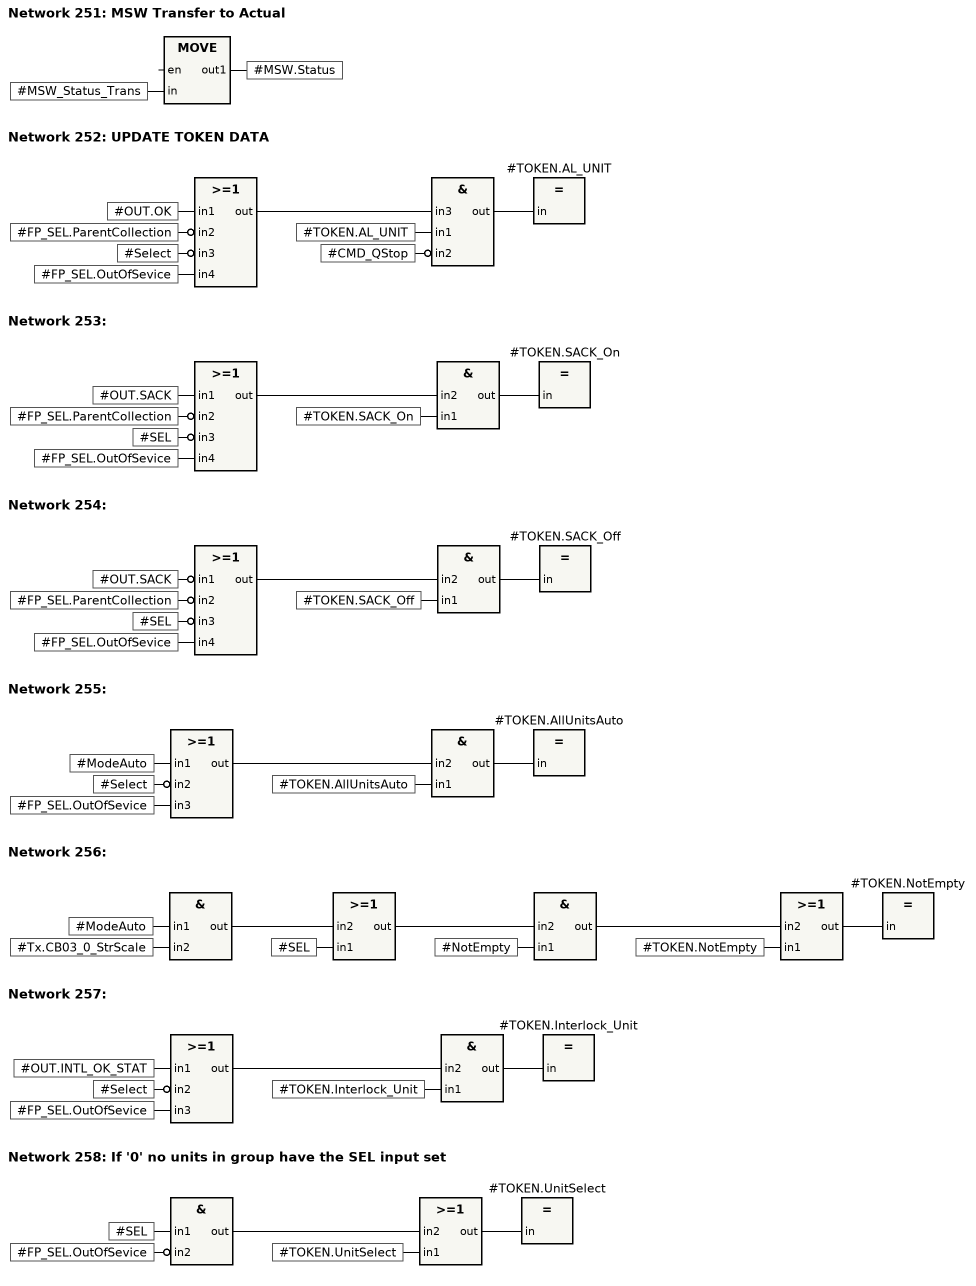
   #MSW.Status := #MSW_Status_Trans;
END_REGION

REGION Network 252: UPDATE TOKEN DATA
   #TOKEN.AL_UNIT := (#OUT.OK OR NOT #FP_SEL.ParentCollection OR NOT #Select OR #FP_SEL.OutOfSevice) AND #TOKEN.AL_UNIT AND NOT #CMD_QStop;
END_REGION

REGION Network 253
   // Build 005 - 24.Jun.2020 (MIA-US): Replace "Select" with "SEL"
   #TOKEN.SACK_On := (#OUT.SACK OR NOT #FP_SEL.ParentCollection OR NOT #SEL OR #FP_SEL.OutOfSevice) AND #TOKEN.SACK_On;
END_REGION

REGION Network 254
   #TOKEN.SACK_Off := (NOT #OUT.SACK OR NOT #FP_SEL.ParentCollection OR NOT #SEL OR #FP_SEL.OutOfSevice) AND #TOKEN.SACK_Off;
END_REGION

REGION Network 255
   #TOKEN.AllUnitsAuto := (#ModeAuto OR NOT #Select OR #FP_SEL.OutOfSevice) AND #TOKEN.AllUnitsAuto;
END_REGION

REGION Network 256
   #TOKEN.NotEmpty := (((#ModeAuto AND #Tx.CB03_0_StrScale) OR #SEL) AND #NotEmpty) OR #TOKEN.NotEmpty;
END_REGION

REGION Network 257
   #TOKEN.Interlock_Unit := (#OUT.INTL_OK_STAT OR NOT #Select OR #FP_SEL.OutOfSevice) AND #TOKEN.Interlock_Unit;
END_REGION

REGION Network 258: If '0' no units in group have the SEL input set
   #TOKEN.UnitSelect := (#SEL AND NOT #FP_SEL.OutOfSevice) OR #TOKEN.UnitSelect;
END_REGION

REGION Network 259: Start Warning
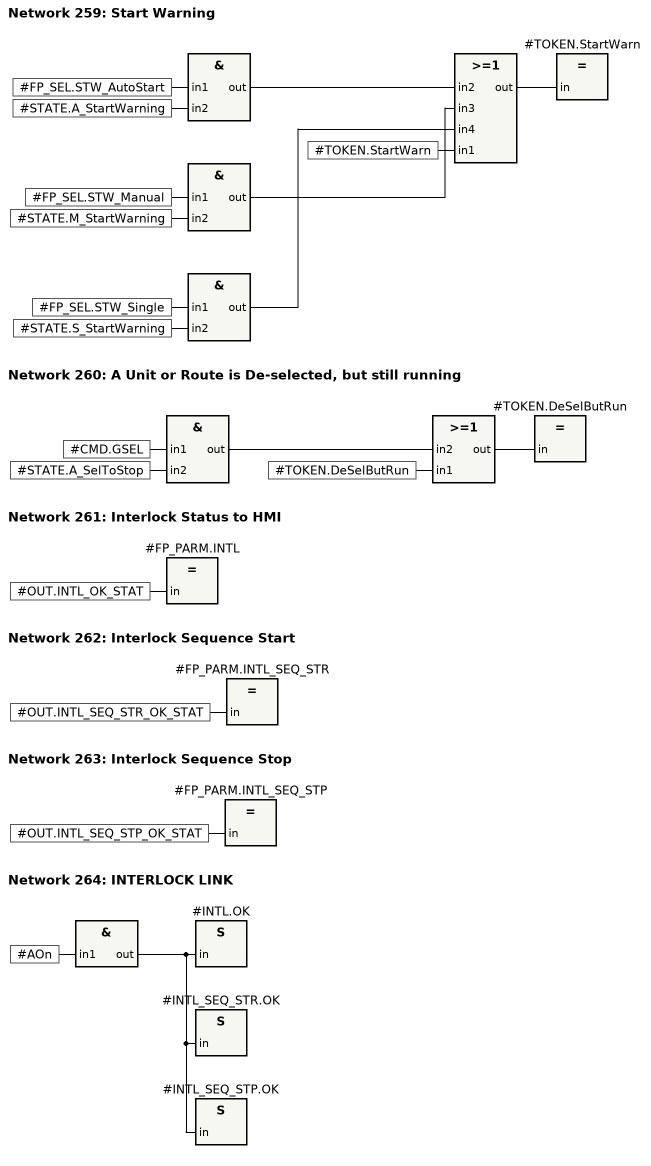
   #TOKEN.StartWarn := (#FP_SEL.STW_AutoStart AND #STATE.A_StartWarning) OR (#FP_SEL.STW_Manual AND #STATE.M_StartWarning) OR (#FP_SEL.STW_Single AND #STATE.S_StartWarning) OR #TOKEN.StartWarn;
END_REGION

REGION Network 260: A Unit or Route is De-selected, but still running
   #TOKEN.DeSelButRun := (#CMD.GSEL AND #STATE.A_SelToStop) OR #TOKEN.DeSelButRun;
END_REGION

REGION Network 261: Interlock Status to HMI
   #FP_PARM.INTL := #OUT.INTL_OK_STAT;
END_REGION

REGION Network 262: Interlock Sequence Start
   #FP_PARM.INTL_SEQ_STR := #OUT.INTL_SEQ_STR_OK_STAT;
END_REGION

REGION Network 263: Interlock Sequence Stop
   #FP_PARM.INTL_SEQ_STP := #OUT.INTL_SEQ_STP_OK_STAT;
END_REGION

REGION Network 264: INTERLOCK LINK
   IF #AOn THEN
       #INTL.OK := TRUE;
       #INTL_SEQ_STR.OK := TRUE;
       #INTL_SEQ_STP.OK := TRUE;
   END_IF;
END_REGION

REGION Network 265: Bit 1: Detect first occuring interlock, unit running
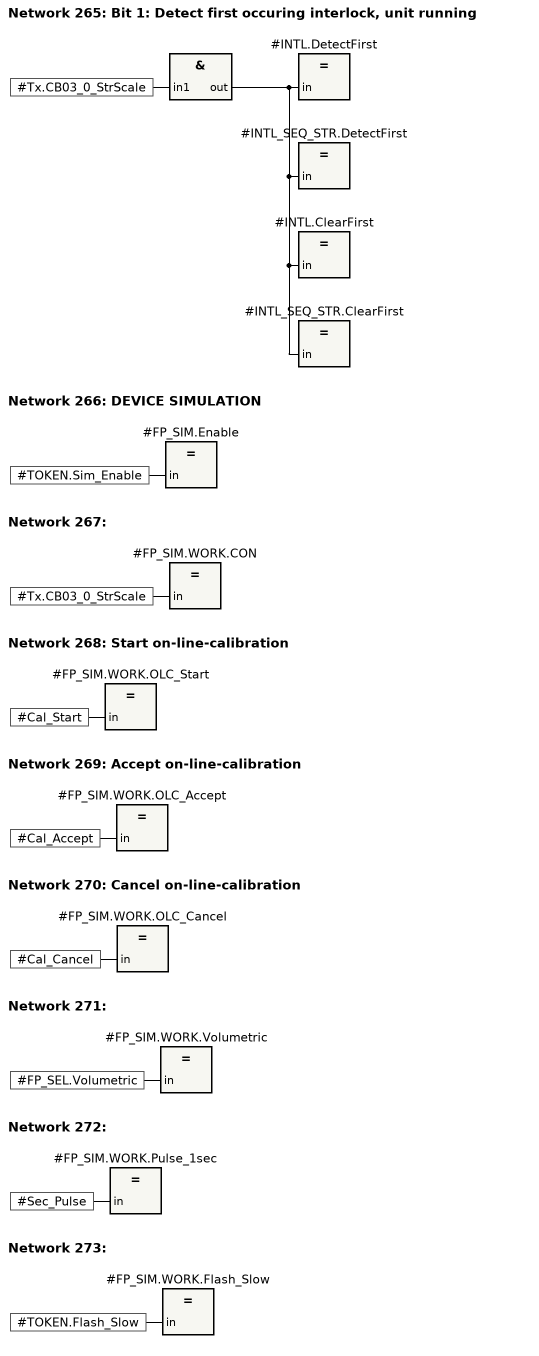
   #INTL.DetectFirst := #Tx.CB03_0_StrScale;
   #INTL_SEQ_STR.DetectFirst := #Tx.CB03_0_StrScale;
   #INTL.ClearFirst := #Tx.CB03_0_StrScale;
   #INTL_SEQ_STR.ClearFirst := #Tx.CB03_0_StrScale;
END_REGION

REGION Network 266: DEVICE SIMULATION
   #FP_SIM.Enable := #TOKEN.Sim_Enable;
END_REGION

REGION Network 267
   #FP_SIM.WORK.CON := #Tx.CB03_0_StrScale;
END_REGION

REGION Network 268: Start on-line-calibration
   #FP_SIM.WORK.OLC_Start := #Cal_Start;
END_REGION

REGION Network 269: Accept on-line-calibration
   #FP_SIM.WORK.OLC_Accept := #Cal_Accept;
END_REGION

REGION Network 270: Cancel on-line-calibration
   #FP_SIM.WORK.OLC_Cancel := #Cal_Cancel;
END_REGION

REGION Network 271
   #FP_SIM.WORK.Volumetric := #FP_SEL.Volumetric;
END_REGION

REGION Network 272
   #FP_SIM.WORK.Pulse_1sec := #Sec_Pulse;
END_REGION

REGION Network 273
   #FP_SIM.WORK.Flash_Slow := #TOKEN.Flash_Slow;
END_REGION

REGION Network 274: Write STAT to OUT
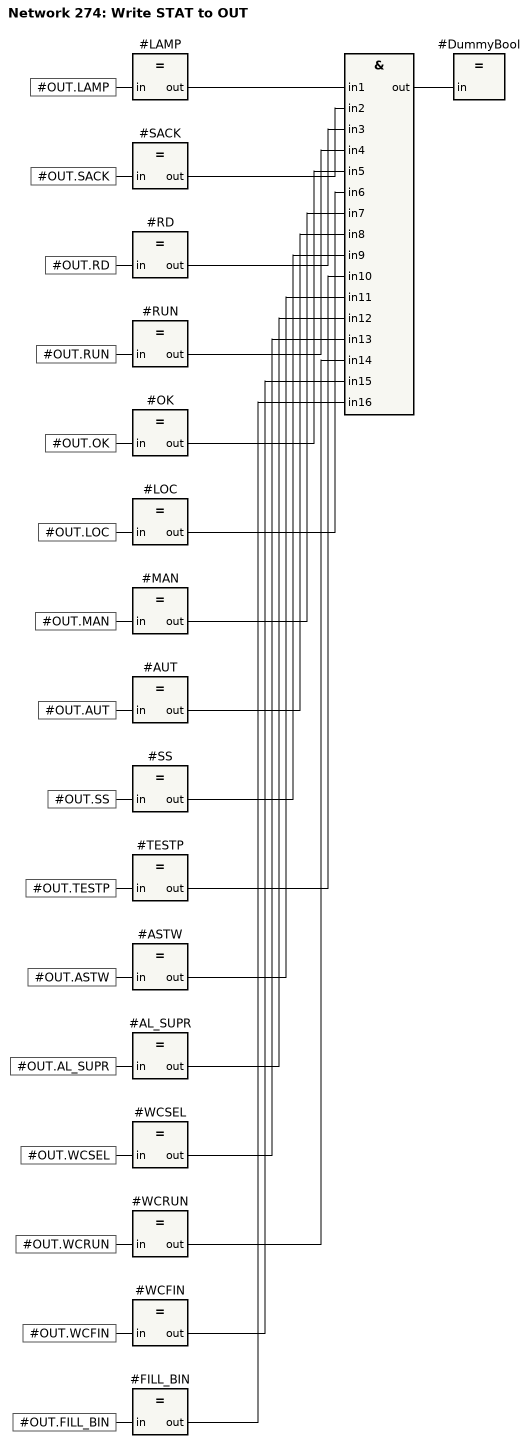
   #LAMP := #OUT.LAMP;
   #SACK := #OUT.SACK;
   #RD := #OUT.RD;
   #RUN := #OUT.RUN;
   #OK := #OUT.OK;
   #LOC := #OUT.LOC;
   #MAN := #OUT.MAN;
   #AUT := #OUT.AUT;
   #SS := #OUT.SS;
   #TESTP := #OUT.TESTP;
   #ASTW := #OUT.ASTW;
   #AL_SUPR := #OUT.AL_SUPR;
   #WCSEL := #OUT.WCSEL;
   #WCRUN := #OUT.WCRUN;
   #WCFIN := #OUT.WCFIN;
   #FILL_BIN := #OUT.FILL_BIN;
   #DummyBool := #OUT.LAMP AND #OUT.SACK AND #OUT.RD AND #OUT.RUN AND #OUT.OK AND #OUT.LOC AND #OUT.MAN AND #OUT.AUT AND #OUT.SS AND #OUT.TESTP AND #OUT.ASTW AND #OUT.AL_SUPR AND #OUT.WCSEL AND #OUT.WCRUN AND #OUT.WCFIN AND #OUT.FILL_BIN;
END_REGION
END_FUNCTION_BLOCK

FUNCTION_BLOCK "ACESYS_PFISTER"   // FB216, FBD
TITLE = ACESYS V8.0 - Build 007 - PFISTER Block
{ S7_Optimized_Access := 'FALSE' }
AUTHOR : FLSmidth
FAMILY : ACESYS
NAME : PFISTER
VERSION : 8.0
// Pfister Block
   VAR_INPUT
      CMD : "ACESYS_GRP_CMD";
      INREF : Int;   // Address reference for Input data
      OUTREF : Int;   // Address reference for Output data
      NET : Int;   // Net number
      NODE : Int;   // Node Number
      FUNCTYPE : Int;   // Function Type
      OPTIONS : Int;   // Operation Options
      SEL : Bool := TRUE;   // Unit Select by User program
      ASTR : Bool := TRUE;   // Auto Start
      SSW : Bool := TRUE;   // Safety Switch
      FSTOP : Bool;   // Filling Devices stopped
      AERA_SILO : Bool;   // Release Aeration Silo
      AERA_PREH : Bool;   // Release Aeration Prehopper
      GAS_SILO : Bool;   // Select Aeration with Gas Silo
      GAS_PREH : Bool;   // Select Aeration with Gas Prehopper
      TOT1_RES : Bool;   // Reset Totalizer 1
      TOT2_RES : Bool;   // Reset Totalizer 2
      SP : Real;   // Feed setpoint
   END_VAR
   VAR_OUTPUT
      INTL : "ACESYS_INTL";   // Interlock
      INTL_SEQ_STR : "ACESYS_INTL";   // Interlock Sequence Start
      INTL_SEQ_STP : "ACESYS_INTL";   // Interlock Sequence Stop
      LAMP : Bool;   // Lamp 1
      SACK : Bool;   // Start Acknowledge
      RD : Bool;   // Run delayed 1
      RUN : Bool;   // Run 1
      OK : Bool;   // Unit Status OK (no alarms)
      WARN : Bool;   // Unit Warning ("1" = No Warning Present)
      LOC : Bool;   // Unit in Local Mode
      MAN : Bool;   // Unit in Manual Mode
      AUT : Bool;   // Unit in Auto Mode
      SS : Bool;   // Unit in Single Start Mode
      ASTW : Bool;   // Start warning
      AL_SUPR : Bool;   // Supress Child Alarms
      OLC_SEL : Bool;   // On-line Calibration Selected
      OLC_RUN : Bool;   // On-line Calibration Active
      OLC_FIN : Bool;   // On-line Calibration Finished
      OLC_ACC : Bool;   // On-line Calibration Accepted
      CORR_Pct : Real;   // Acutal Coorrection converted Percent
      FEED_Pct : Real;   // Actual Feed converted Percent
      FEED_Eng : Real;   // Actual Feed converted Eng.units
      WEIGHT_Pct : Real;   // Actual Bin Weight converted Percent
      WEIGHT_Eng : Real;   // Actual Bin Weight converted Eng.Units
      WSP_Pct : Real;   // Actual Working Set Point Percent
      WSP_Eng : Real;   // Actual Working Set Point Eng. Units
      SPEED_Eng : Real;   // Actual Speed Prefeeder (rpm)
      SP_Pct : Real;   // Set Point to Feeder converted Percent
      SP_Eng : Real;   // Set Point to Feeder converted Eng.Units
      TOTAL_1 : Real;   // Totalizer 1 (t)
      TOTAL_2 : Real;   // Totalizer 2 (t)
      MSW : "ACESYS_HMI_STAT_32T";
   END_VAR
   VAR_IN_OUT
      TOKEN : "ACESYS_TOKEN";
   END_VAR
   VAR
      BlockInfo : Struct
         Ace_Version : Int;   // Acesys Block Version Number
         Ace_BuildNo : Int;   // Acesys Block Build Number
         State_Act : Int;   // Actual State Number
         State_Prev : Int;   // Previous State Number
         DB_Number : Int;   // Block Instance DB Number
      END_STRUCT;
      FP_CMD : Struct   // Faceplate Commands
         QuickStop : Bool;
         StartOLC : Bool;
         StopOLC : Bool;
         IgnoreResult : Bool;
         AcceptResult : Bool;
         SetUserCorr : Bool;
         Spare_14 : Bool;
         AckAlarm : Bool;
         Auto : Bool;
         Manual : Bool;
         Local : Bool;
         Start : Bool;
         Reset : Bool;
         Stop : Bool;
         ResetTot1 : Bool;
         ResetTot2 : Bool;
      END_STRUCT;
      FP_SEL : Struct   // Faceplate Selections
         STW_AutoStart : Bool;   // Faceplate Start Warning in Auto Start mode
         STW_Manual : Bool;   // Faceplate Start Warning in Manual mode
         STW_Single : Bool;   // Faceplate Start Warning in Single Start mode
         ParentSupress : Bool;   // Enable Parent Supress of alarms
         ParentCollection : Bool;   // Enable Parent Collection
         INCH_Man : Bool;   // Enable Inching in Manual Mode
         OutOfSevice : Bool;   // Select Out of Service
         WarningDrive : Bool;   // 0 = Failure Drive / 1 = Warning Drive
         Spare7 : Bool;
         Spare6 : Bool;
         Spare5 : Bool;
         Spare4 : Bool;
         Spare3 : Bool;
         Spare2 : Bool;
         Spare1 : Bool;
      END_STRUCT;
      FP_EN : Struct
         Mode_Auto : Bool;
         Mode_Man : Bool;
         Mode_Loc : Bool;
         Mode_Test : Bool;
         Mode_SS_Field : Bool;
         Mode_SS_FP : Bool;
         PB_QStop : Bool;
         Aeration_Silo_Const : Bool;
         Aeration_PreH_Const : Bool;
         Volumetric_Feeder : Bool;
         Volumetric_PreFeeder : Bool;
         Volumetric_Refilling : Bool;
         Empty_Next : Bool;
         Empty_All : Bool;
         TOT1_FP_Reset : Bool;   // Enable Reset Totalizer 1 from Faceplate
         TOT2_FP_Reset : Bool;   // Enable Reset Totalizer 2 from Faceplate
      END_STRUCT;
      FP_DIM : Struct   // Faceplate Dimmed Buttons
         Auto : Bool;
         Local : Bool;
         Manual : Bool;
         Start : Bool;
         Stop : Bool;
         QStop : Bool;
         Reset : Bool;
         StartOLC : Bool;
         AcceptResult : Bool;
         CancelResult : Bool;
         StopOLC : Bool;
         SetUserCorr : Bool;
         ResetTot1 : Bool;
         ResetTot2 : Bool;
         Spare9 : Bool;
         Spare8 : Bool;
         Spare7 : Bool;
         Spare6 : Bool;
         Spare5 : Bool;
         Spare4 : Bool;
         Spare3 : Bool;
         Spare2 : Bool;
         Spare1 : Bool;
      END_STRUCT;
      FP_SHOW : Struct   // Faceplate Show Buttons
         PB_Auto : Bool;
         PB_Local : Bool;
         PB_Manual : Bool;
         PB_Start : Bool;
         PB_Stop : Bool;
         PB_QStop : Bool;
         ACK : Bool;
         PB_Reset : Bool;
         ASTR : Bool;
         SSW : Bool;
         Spare06 : Bool;
         Spare05 : Bool;
         Spare04 : Bool;
         Spare03 : Bool;
         Spare02 : Bool;
         Spare01 : Bool;
      END_STRUCT;
      FP_PARM : Struct   // Faceplate Parameters
         StartWarn_Pre : Int := 15;
         StartWarn_Acc : Int;
         RunDelay_Pre : Int := 3;
         RunDelay_Acc : Int;
         DelayStart_Pre : Int := 3;
         DelayStart_Acc : Int;
         DelayStop_Pre : Int;
         DelayStop_Acc : Int;
         ReturnMon_Pre : Int := 3;
         ReturnMon_Acc : Int;
         StopReason : Int;
         CORR_User : Real;
         SpeedSP_Feeder : Real;
         SpeedSP_PreFeeder : Real;
         SpeedSP_Refilling : Real;
         INTL : Bool;   // Interlock
         INTL_SEQ_STR : Bool;   // Interlock Sequence Start
         INTL_SEQ_STP : Bool;   // Interlock Sequence Stop
         Spare13 : Bool;
         Spare12 : Bool;
         Spare11 : Bool;
         Spare10 : Bool;
         Spare09 : Bool;
         Spare08 : Bool;
         Spare07 : Bool;
         Spare06 : Bool;
         Spare05 : Bool;
         Spare04 : Bool;
         Spare03 : Bool;
         Spare02 : Bool;
         Spare01 : Bool;
      END_STRUCT;
      Rx : Struct
         ServiceID : Byte := BYTE#16#01;   // Insignificant,from write protocol
         AdministrationNo : Byte;   // Number from write protocol
         ProtocolNo : Byte := BYTE#16#14;   // Protocol must be 20 !!!
         NodeNo : Byte;   // Node number
         HostAddress : DWord;   // Network address of host system = client
         ErrorDevice : DInt;   // ERR Device indicating error
         PresentError : DInt;   // ERR Error number
         StF_24 : Bool;   // StF_24 Status Feeder Bit 24
         StF_25 : Bool;   // StF_25
         StF_26 : Bool;   // StF_26
         StF_27 : Bool;   // StF_27
         StF_28 : Bool;   // StF_28
         StF_29 : Bool;   // StF_29
         StF_30 : Bool;   // StF_30
         StF_31 : Bool;   // StF_31
         FeederSlideGateFault : Bool;   // StF_16 Slide gate above feeder is not in required position
         FeederSlideGateOpen : Bool;   // StF_17 Slide gate above feeder is open
         PrefeederFault : Bool;   // StF_18 Fault of prefeeder
         PrefeederRunning : Bool;   // StF_19 Prefeeder is running
         LoadingQuantityReached : Bool;   // StF_20 Loading cycle finished (only with loading application)
         StF_21 : Bool;   // StF_21 Status Feeder Bit 21
         StF_22 : Bool;   // StF_22
         StF_23 : Bool;   // StF_23
         FaultFeeder : Bool;   // StF_08 Fault of feeder
         FeedingStarted : Bool;   // StF_09 Feeder is in operation
         RunningBackward : Bool;   // StF_10 Direction of feeder drive = backward
         RunningForward : Bool;   // StF_11 Direction of feeder drive = forward (feeding direction)
         LoadingAboveLowerLimit : Bool;   // StF_12 Loading of feeder higher than low level WL1
         LoadingAboveUpperLimit : Bool;   // StF_13 Loading of feeder higher than high level WH1
         LoadingBelowEmptyLimit : Bool;   // StF_14 Loading of feeder lower than empty WLL1
         FeederSlideGateClosed : Bool;   // StF_15 Slide gate above feeder is closed
         ControlVoltageOK : Bool;   // StF_00 Control voltage generation in cabinet is ok
         NotEmergencyStop : Bool;   // StF_01 Emergency stop hardwired input is not active
         StartIsReleased : Bool;   // StF_02 Start is released via hardwired input
         AutomaticMode : Bool;   // StF_03 Feeder is in Remote (valid also in volumetric mode). Ctrl only via PCS
         FieldMode : Bool;   // StF_04 Feeder is in Field mode. Control only via FLP
         LocalMode : Bool;   // StF_05 Feeder is in Local mode. Control via panel and/orFLP
         VolumetricModeActive : Bool;   // StF_06 Volumetric mode is selected for one of the drives
         AdjustModeActive : Bool;   // StF_07 For service purposes speed is freezed as long as this signal is high
         SiloAerationActive : Bool;   // StB_24 Aeration in silo cone is released
         SiloAerationFault : Bool;   // StB_25 Aeration in silo cone is faulty (power to valves)
         RefillSlideGateClosed : Bool;   // StB_26 Slide gate above prehopper is closed
         RefillSlideGateFault : Bool;   // StB_27 Fault in slide gate sequence
         RefillSlideGateOpen : Bool;   // StB_28 Slide gate above prehopper is open
         StB_29 : Bool;   // StB_29 Status Bins Bit 29
         StB_30 : Bool;   // StB_30
         StB_31 : Bool;   // StB_31
         FlapGateClosed : Bool;   // StB_16 Flap above prehopper is closed
         FlapGateFault : Bool;   // StB_17 Fault in flap sequence
         FlapGateOpen : Bool;   // StB_18 Flap above prehopper is open
         SiloLevelAboveHighLimit : Bool;   // StB_19 Level in silo higher than high level
         SiloLevelAboveMaximum : Bool;   // StB_20 Level in silo higher than max level
         SiloLevelBelowLowerLimit : Bool;   // StB_21 Level in silo lower than low level
         SiloLevelBelowMinimum : Bool;   // StB_22 Level in silo lower than min level
         SiloLevelFault : Bool;   // StB_23 Fault in silo level measurement
         OLCFault : Bool;   // StB_08 Fault in online calibration
         OLCFinished : Bool;   // StB_09 Online calibration has finished
         OLCRunning : Bool;   // StB_10 Online calibration is in operation
         OLCStarted : Bool;   // StB_11 Online calibration has started
         AgitatorFault : Bool;   // StB_12 Fault in agitator sequence
         AgitatorRunning : Bool;   // StB_13 Agitator is in operation
         RefillingFault : Bool;   // StB_14 Fault in refilling sequence
         RefillingRunning : Bool;   // StB_15 Refilling of prehopper is in operation
         PreHLevelAboveHighLimit : Bool;   // StB_00 Level in prehopper higher than high level. OLC can be started
         PreHLevelAboveMaximum : Bool;   // StB_01 Level in prehopper higher than max level. Refilling will be aborted
         PreHLevelBelowLowerLimit : Bool;   // StB_02 Level in prehopper lower than low level. OLC will be aborted
         PreHLevelBelowMinimum : Bool;   // StB_03 Level in prehopper lower than min level. Feeding will be influenced
         PreHLevelFault : Bool;   // StB_04 Fault in prehopper level measurement
         PreHLevelMaxProbe : Bool;   // StB_05 Max probe has detected volumetric max level(Recalculation level limits)
         PreHAerationActive : Bool;   // StB_06 Aeration in prehopper cone is released
         PreHAerationFault : Bool;   // StB_07 Aeration in prehopper cone is faulty (power to valves)
         Feedrate : Real;   // FI1 Real feed rate
         SpeedWeighFeederDrive : Real;   // SI1 Real speed of feeder
         RelativeLoadAtDischarge : Real;   // WI1a Real load of feeder relative to nominal load
         Totalizer1 : Real;   // FQ1 Short time integral of real feed rate
         PrehopperLevel : Real;   // LI3 Level in Prehopper as weight
         DifferenceOfOLC : Real;   // WD1 Difference of fed quantity FQ3 and weighed quantity WI3
         Optional1_Feeder_Config : Struct   // Optional read value as selected in write table
            SlideGateFeeder_Present : Bool;   // Feeder config - bit 24
            SlideGateFeeder_25 : Bool;   // Feeder config - bit 25
            SlideGateFeeder_26 : Bool;   // Feeder config - bit 26
            SlideGateFeeder_27 : Bool;   // Feeder config - bit 27
            NotUsed_28 : Bool;   // Feeder config - bit 28
            NotUsed_29 : Bool;   // Feeder config - bit 29
            NotUsed_30 : Bool;   // Feeder config - bit 30
            NotUsed_31 : Bool;   // Feeder config - bit 31
            Prefeeder_Present : Bool;   // Feeder config - bit 16
            Prefeeder_17 : Bool;   // Feeder config - bit 17
            Prefeeder_18 : Bool;   // Feeder config - bit 18
            Prefeeder_19 : Bool;   // Feeder config - bit 19
            PreMeasurement_Present : Bool;   // Feeder config - bit 20
            PreMeasurement_21 : Bool;   // Feeder config - bit 21
            PreMeasurement_22 : Bool;   // Feeder config - bit 22
            PreMeasurement_23 : Bool;   // Feeder config - bit 23
            Internal_08 : Bool;   // Feeder config - bit 8
            Internal_09 : Bool;   // Feeder config - bit 9
            Internal_10 : Bool;   // Feeder config - bit 10
            Internal_11 : Bool;   // Feeder config - bit 11
            Internal_12 : Bool;   // Feeder config - bit 12
            Internal_13 : Bool;   // Feeder config - bit 13
            Internal_14 : Bool;   // Feeder config - bit 14
            Internal_15 : Bool;   // Feeder config - bit 15
            FeederType_1 : Bool;   // Feeder config - bit 0
            FeederType_2 : Bool;   // Feeder config - bit 1
            FeederType_3 : Bool;   // Feeder config - bit 2
            FeederType_4 : Bool;   // Feeder config - bit 3
            NotUsed_04 : Bool;   // Feeder config - bit 4
            NotUsed_05 : Bool;   // Feeder config - bit 5
            NotUsed_06 : Bool;   // Feeder config - bit 6
            NotUsed_07 : Bool;   // Feeder config - bit 7
         END_STRUCT;
         Optional2_PreH_Config : Struct   // Optional read value as selected in write table
            Refilling_Present : Bool;   // Prehopper config - bit 24
            Agitator_25 : Bool;   // Prehopper config - bit 25
            Agitator_26 : Bool;   // Prehopper config - bit 26
            Agitator_27 : Bool;   // Prehopper config - bit 27
            SlideGatePreH_Present : Bool;   // Prehopper config - bit 28
            SlideGatePreH_29 : Bool;   // Prehopper config - bit 29
            SlideGatePreH_30 : Bool;   // Prehopper config - bit 30
            SlideGatePreH_31 : Bool;   // Prehopper config - bit 31
            PreHopAeration_Present : Bool;   // Prehopper config - bit 16
            PreHopAeration_17 : Bool;   // Prehopper config - bit 17
            PreHopAeration_18 : Bool;   // Prehopper config - bit 18
            PreHopAeration_19 : Bool;   // Prehopper config - bit 19
            Agitator_Present : Bool;   // Prehopper config - bit 20
            Agitator_21 : Bool;   // Prehopper config - bit 21
            Agitator_22 : Bool;   // Prehopper config - bit 22
            Agitator_23 : Bool;   // Prehopper config - bit 23
            PressCompensate_Present : Bool;   // Prehopper config - bit 8
            PressCompensate_09 : Bool;   // Prehopper config - bit 9
            PressCompensate_10 : Bool;   // Prehopper config - bit 10
            PressCompensate_11 : Bool;   // Prehopper config - bit 11
            NotUsed_12 : Bool;   // Prehopper config - bit 12
            NotUsed_13 : Bool;   // Prehopper config - bit 13
            NotUsed_14 : Bool;   // Prehopper config - bit 14
            NotUsed_15 : Bool;   // Prehopper config - bit 15
            PreHopper_Present : Bool;   // Prehopper config - bit 0
            Prehopper_01 : Bool;   // Prehopper config - bit 1
            Prehopper_02 : Bool;   // Prehopper config - bit 2
            Prehopper_03 : Bool;   // Prehopper config - bit 3
            BlockSystem_Present : Bool;   // Prehopper config - bit 4
            BlockSystem_05 : Bool;   // Prehopper config - bit 5
            BlockSystem_06 : Bool;   // Prehopper config - bit 6
            BlockSystem_07 : Bool;   // Prehopper config - bit 7
         END_STRUCT;
         Optional3_Firmware : Struct   // Optional read value as selected in write table
            Firmware_4 : Byte;
            Firmware_3 : Byte;
            Firmware_2 : Byte;
            Firmware_1 : Byte;
         END_STRUCT;
         Optional4_Range_Feed : Real;   // Optional read value as selected in write table
         PresentCorrectionValue : Real;   // QY1 Result of last online calibration
         CurrentOfFeeder : Real;   // II1 Real current of feeder motor
         LoadAtDischarge : Real;   // WI1a Real load of feeder at discharge
         RelativeLoadAtMeasuring : Real;   // WI1 Relative loading at measuring related to nominal load
         Totalizer2 : Real;   // FQ2 Long time integral of real feed rate
         CurrentOfPrefeeder : Real;   // II2 Real current of prefeeder motor
         SetpointOfPrefeeder : Real;   // SY2/GY2 Real speed (position) setpoint to prefeeder drive
         FeedbackOfPrefeeder : Real;   // SI2/GI2 Real speed (position) of prefeeder
         CurrentOfRefilling : Real;   // II3 Real current of refilling motor
         SetpointOfRefilling : Real;   // SY3/GY3 Real speed (position) setpoint to refilling drive
         FeedbackOfRefilling : Real;   // SI3/GI3 Real speed (position) of refilling
         LevelOfMaterialInSilo : Real;   // LI4 Level in silo as weight
         Optional5_Range_Prehoppe : Real;   // Optional read value as selected in write table
         Optional6_WSP_Eng : Real;   // Optional read value as selected in write table
         Optional7_Total_OLC : Real;   // Optional read value as selected in write table
         Optional8_Spare : Real;   // Optional read value as selected in write table
      END_STRUCT;
      Tx : Struct
         ServiceID : Byte;   // Insignificant, number is returned in read protocol
         AdministrationNo : Byte;   // Number is returned in read protocol
         ProtocolNo : Byte := BYTE#16#14;   // Protocol must be 20 !!!
         NodeNo : Byte;   // Node number
         NDY : DWord;   // Not defined yet
         Cmd_24 : Bool;   // Command Bit 24
         Cmd_25 : Bool;   // Cmd_25
         Cmd_26 : Bool;   // Cmd_26
         Cmd_27 : Bool;   // Cmd_27
         Cmd_28 : Bool;   // Cmd_28
         Cmd_29 : Bool;   // Cmd_29
         Cmd_30 : Bool;   // Cmd_30
         Cmd_31 : Bool;   // Cmd_31
         StopOnlineCalibration : Bool;   // Cmd_16 Stop online calibration in remote mode
         VolumetricModeRefilling : Bool;   // Cmd_17 Set feeder refilling drive to volumetric mode (speed setpoint SY3r)
         RefillingOfPreHStopper : Bool;   // Cmd_18 Feedback from refill drive. Precondition for online calibration.
         ReleaseSiloAeration : Bool;   // Cmd_19 General release of aeration
         SiloAerationPermanent : Bool;   // Cmd_20 Aeration is operated permanently instead of cyclewise (air or gas)
         SiloAerationSelectionAir : Bool;   // Cmd_21 Selection of aeration media to normal air. Off = inert gas
         Cmd_22 : Bool;   // Cmd_22
         Cmd_23 : Bool;   // Cmd_23
         VolumetricModeFeeder : Bool;   // Cmd_08 Set feeder drive to volumetric mode (speed setpoint SY1r)
         VolumetricModePrefeeder : Bool;   // Cmd_09 Set prefeeder drive to volumetric mode (speed setpoint SY2r)
         AcceptRemoteZeroCorr : Bool;   // Cmd_10 Acceptance of correction value sent from plant control
         AcceptZeroCorrection : Bool;   // Cmd_11 Acceptance of result (= correction value) of online calibration
         PreHAerationPermanent : Bool;   // Cmd_12 Aeration is operated permanently instead of cyclewise (air or gas)
         PreHAerationSelectionAir : Bool;   // Cmd_13 Selection of aeration media to normal air. Off = inert gas
         ReleasePrehopperAeration : Bool;   // Cmd_14 General release of aeration
         StartOnlineCalibration : Bool;   // Cmd_15 Start online calibration in remote mode
         AcknowledgeFailure : Bool;   // Cmd_00 Reset error messages
         EmpySystem : Bool;   // Cmd_01 Prehopper refilling is stopped and feeding station runs empty
         RemoteOn : Bool;   // Cmd_02 Remote = full control of feeder from PCS
         EnableEmpyFeeder : Bool;   // Cmd_03 With next "stop feeding " cmd feeder will run till empty and then stop
         ResetTotalizer1 : Bool;   // Cmd_04 Reset totalizer-1 (FQ1)
         ResetTotalizer2 : Bool;   // Cmd_05 Reset totalizer-2 (FQ2)
         StartFeeding : Bool;   // Cmd_06 Start feeder in remote operation
         StopFeeding : Bool;   // Cmd_07 Stop feeder in remote operation
         E160 : Bool;   // E160 Reserved commands CMDr
         E161 : Bool;   // E161
         E162 : Bool;   // E162
         E163 : Bool;   // E163
         E164 : Bool;   // E164
         E165 : Bool;   // E165
         E166 : Bool;   // E166
         E167 : Bool;   // E167
         E150 : Bool;   // E150
         E151 : Bool;   // E151
         E152 : Bool;   // E152
         E153 : Bool;   // E153
         E154 : Bool;   // E154
         E155 : Bool;   // E155
         E156 : Bool;   // E156
         E157 : Bool;   // E157
         E140 : Bool;   // E140
         E141 : Bool;   // E141
         E142 : Bool;   // E142
         E143 : Bool;   // E143
         E144 : Bool;   // E144
         E145 : Bool;   // E145
         E146 : Bool;   // E146
         E147 : Bool;   // E147
         E130 : Bool;   // E130
         E131 : Bool;   // E131
         E132 : Bool;   // E132
         E133 : Bool;   // E133
         E134 : Bool;   // E134
         E135 : Bool;   // E135
         E136 : Bool;   // E136
         E137 : Bool;   // E137
         SetpointOfFeedrate : Real;   // FY1 feedrate setpoint used in remote mode
         RemoteCorrection : Real;   // QY1r Correction of zero sent from plant control. To be made valid by command
         SetpointLoadingQuantity : Real;   // QYL Loading mass setpoint (used for loading operations)
         SpeedSetpFeederDrive : Real;   // SY1r Speed setpoint valid in volumetric mode for feeder drive
         SpeedSetpPrefeederDrive : Real;   // SY2r Speed setpoint valid in volumetric mode for prefeeder drive
         SpeedSetpRefillingDrive : Real;   // SY3r Speed setpoint valid in volumetric mode for refilling drive
         FreeValue1 : Real;   // Not yet defined
         FreeValue2 : Real;   // Not yet defined
         VAR53 : Real;   // Reserved value VAR53
         VAR59 : Real;   // Reserved value VAR59
         SelectOptionalReadVal1 : Byte;   // Number of optional read value
         SelectOptionalReadVal2 : Byte;   // Number of optional read value
         SelectOptionalReadVal3 : Byte;   // Number of optional read value
         SelectOptionalReadVal4 : Byte;   // Number of optional read value
         SelectOptionalReadVal5 : Byte;   // Number of optional read value
         SelectOptionalReadVal6 : Byte;   // Number of optional read value
         SelectOptionalReadVal7 : Byte;   // Number of optional read value
         SelectOptionalReadVal8 : Byte;   // Number of optional read value
      END_STRUCT;
      FP_SIM : "ACESYS_SIM_PFISTER";
      STATE : Struct
         A_AutoStart : Bool;
         A_DelayedStart : Bool;
         A_DelayedStop : Bool;
         A_Running : Bool;
         A_Selected : Bool;
         A_SelToStop : Bool;
         A_Stopping : Bool;
         A_SeqStart : Bool;
         A_SeqStop : Bool;
         A_Starting : Bool;
         A_StartWarning : Bool;
         A_Stopped : Bool;
         A_EmptyingSystem : Bool;
         S_AutoStart : Bool;
         S_Running : Bool;
         S_Starting : Bool;
         S_StartWarning : Bool;
         S_Stopped : Bool;
         S_Stopping : Bool;
         S_EmptyingSystem : Bool;
         M_Running : Bool;
         M_Starting : Bool;
         M_StartWarning : Bool;
         M_Stopped : Bool;
         M_Stopping : Bool;
         M_EmptyingSystem : Bool;
         L_Running : Bool;
         L_Stopped : Bool;
         Alarm : Bool;
         Interlock : Bool;
         EmergencyStop : Bool;
         OutOfService : Bool;
      END_STRUCT;
      ONS : Struct
         AckAlarm : Bool;
         Cmd_Auto : Bool;
         Cmd_Manual : Bool;
         CMD_Local : Bool;
         GLTP : Bool;
         CMD_Start : Bool;
         FP_Start_CMD : Bool;
         SecPulse1 : Bool;
         SecPulse2 : Bool;
         Empty_Next : Bool;
         OLCRunning : Bool;
         OLCStarted : Bool;
         TOT1_RES : Bool;
         TOT2_RES : Bool;
         StartOLC : Bool;
         StopOLC : Bool;
         IgnoreResult : Bool;
         AcceptResult : Bool;
         SetUserCorr : Bool;
         ResetTot1 : Bool;
         ResetTot2 : Bool;
         Reset : Bool;
         Spare02 : Bool;
         Spare01 : Bool;
      END_STRUCT;
      StatusWork : Int;
      ModePointer : Int;
      AlarmNo : Int;
      AlarmNo_Old : Int;
      StartWarn_Mem : Int;
      RunDelay_Mem : Int;
      DelayStart_Mem : Int;
      DelayStop_Mem : Int;
      ReturnMon_Mem : Int;
      Watchdog_Mem : Int;
      RET_VAL_Output : Int;
      RET_VAL_Input : Int;
      FeederType : Int;
      TimerAccept_Mem : Int;
      TimerCancel_Mem : Int;
      TimerUserCorr_Mem : Int;
      TimerResetTot1_Mem : Int;
      TimerResetTot2_Mem : Int;
      TimerResetAlarm_Mem : Int;
      ModeAuto : Bool;
      ModeLocal : Bool;
      ModeManual : Bool;
      ModeSingleStart : Bool;
      Select : Bool;   // Parent & Program Select
      CMD_AckAlarm : Bool;
      CMD_Start : Bool;
      CMD_Stop : Bool;
      CMD_QStop : Bool;
      FromStateAuto : Bool;
      FromStateSingle : Bool;
      FromStateManual : Bool;
      FromStateLocal : Bool;
      FromStopState : Bool;
      ALARM_SupressionActive : Bool;
      ALARM_AlarmPresent : Bool;
      ALARM_WarnPresent : Bool;
      ALARM_FailureAckRequired : Bool;
      ALARM_WarnAckRequired : Bool;
      StartWarn_TT : Bool;
      StartWarn_Done : Bool;
      Rundelay_Done : Bool;
      DelayStart_Done : Bool;
      DelayStop_Done : Bool;
      ReturnMon_Done : Bool;
      Trig_RET_ALARM : Bool;
      RET_OneScan : Bool;
      NotEmpty : Bool;   // Unit Stopped un-normal
      Sec_Pulse : Bool;
      Start : Bool;
      Req_Start_OLC : Bool;
      Req_Stop_OLC : Bool;
      OLC_WeightCheckSelLatch : Bool;
      OLC_DeviationFaultMem : Bool;
      OLC_AcceptResult : Bool;
      OLC_CancelResult : Bool;
      OLC_SetUserCorr : Bool;
      OLC_Result_Timer : Bool;
      OLC_AccUserCorr_Timer : Bool;
      ResetTotalizer1 : Bool;
      ResetTotalizer2 : Bool;
      ResetTotalizer1_Timer : Bool;
      ResetTotalizer2_Timer : Bool;
      ResetToPfister : Bool;
      MaxResetTimeDone : Bool;
      OUT : Struct
         LAMP : Bool;
         SACK : Bool;
         RD : Bool;
         RUN : Bool;
         OK : Bool;
         WARN : Bool;
         LOC : Bool;
         MAN : Bool;
         AUT : Bool;
         SS : Bool;
         ASTW : Bool;
         AL_SUPR : Bool;
         OLC_SEL : Bool;
         OLC_RUN : Bool;
         OLC_FIN : Bool;
         OLC_ACC : Bool;
         INTL_OK_STAT : Bool;
         INTL_SEQ_STR_OK_STAT : Bool;
         INTL_SEQ_STP_OK_STAT : Bool;
         MSW_EXT_ALARMFAILUNACK : Bool;
      END_STRUCT;
      MSW_Status_Trans : Int;
   END_VAR
   VAR_TEMP
      AOn : Bool;   // Always On
      AOff : Bool;   // Always Off
      Temp_CON : Bool;
      BusFault : Bool;   // Bus failure
      WatchDog_Elapsed : Bool;
      WatchDog_Same : Bool;
      DummyBool : Bool;
      DummyReal : Real;
      DummyDWord : DWord;
      DummyInt : Int;
      StatPointer_Old : Int;
      StatusBuilder : Int;
      Addr_InstanceDB : DWord;
      Pfister_BlkMove_Len : Int;
      Pfister_Offset : Int;
      DB_Pointer : ANY;
      IO_Pointer : ANY;
      Range_Feed : Real;   // Feed Range (t/h)
      Range_Prehopper : Real;   // Prehopper weighing range (t)
      Status_Add : Int;
      GDC_Pointer : ANY;
      GDC_OptionalValues : Array[0..7] of Byte;
      DummyDint : DInt;
   END_VAR
   VAR_TEMP   // added for the SCL form of the ladder/FBD networks
      _w1 : Bool;
      _w2 : Bool;
      _w3 : Bool;
      _w4 : Bool;
      _w5 : Bool;
      _w6 : Bool;
      _w7 : Bool;
   END_VAR
BEGIN

REGION Network 1: Always On
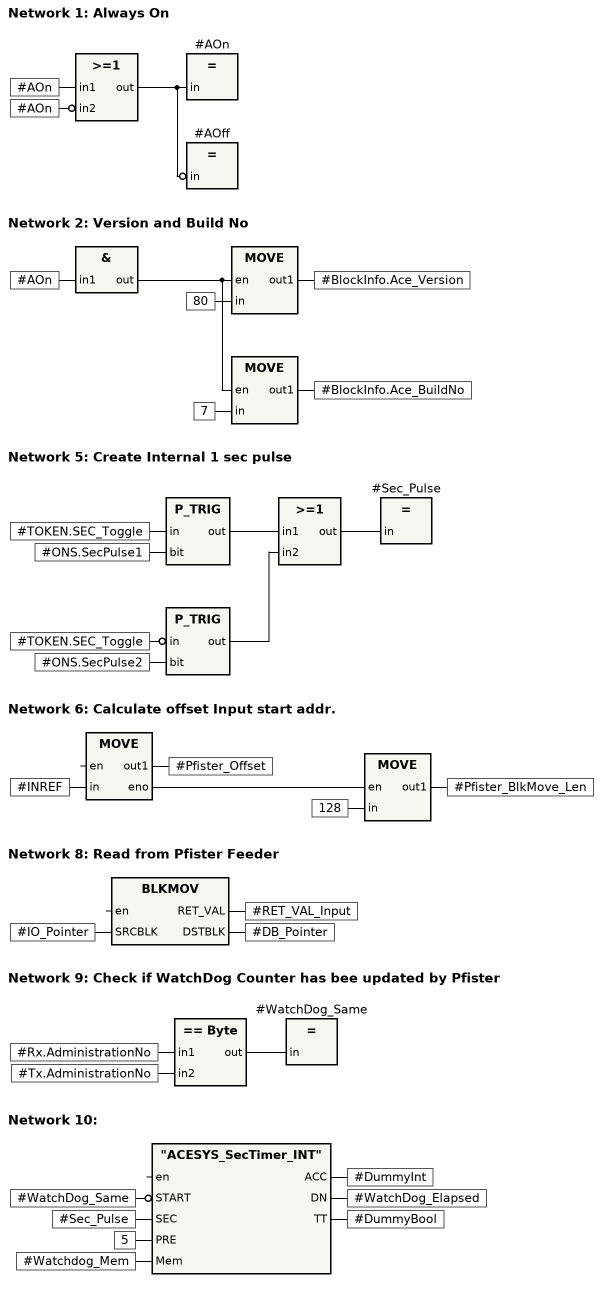
   #AOn := #AOn OR NOT #AOn;
   #AOff := NOT #AOn;
END_REGION

REGION Network 2: Version and Build No
   IF #AOn THEN
       #BlockInfo.Ace_Version := 80;
       #BlockInfo.Ace_BuildNo := 7;
   END_IF;
END_REGION

REGION Network 3 (STL): Instance DB Number to Faceplate
         L     DINO;
         T     #BlockInfo.DB_Number;
END_REGION

REGION Network 4 (SCL): Transfer Interlock OK to Stat
   #OUT.INTL_OK_STAT := PEEK_BOOL(area := 16#84, dbNumber := #BlockInfo.DB_Number, byteOffset := 20, bitOffset := 0);
   #OUT.INTL_SEQ_STR_OK_STAT := PEEK_BOOL(area := 16#84, dbNumber := #BlockInfo.DB_Number, byteOffset := 22, bitOffset := 0);
   #OUT.INTL_SEQ_STP_OK_STAT := PEEK_BOOL(area := 16#84, dbNumber := #BlockInfo.DB_Number, byteOffset := 24, bitOffset := 0);
END_REGION

REGION Network 5: Create Internal 1 sec pulse
   #_w1 := #TOKEN.SEC_Toggle AND NOT #ONS.SecPulse1;   // rising edge
   #ONS.SecPulse1 := #TOKEN.SEC_Toggle;
   #_w2 := NOT #TOKEN.SEC_Toggle AND NOT #ONS.SecPulse2;   // rising edge
   #ONS.SecPulse2 := NOT #TOKEN.SEC_Toggle;
   #Sec_Pulse := #_w1 OR #_w2;
END_REGION

REGION Network 6: Calculate offset Input start addr.
   // Hardware Address
   #Pfister_Offset := #INREF;
   #Pfister_BlkMove_Len := 128;
END_REGION

REGION Network 7 (STL): Target Pointers Recieve input data
         LAR1;  // Make AR1 point to calling program stack
         L     16#10;  // ANY Syntax ID
         T     LB[AR1, P#0.0];  // ..Store Byte 0
         L     16#02;  // Data Type = Byte
         T     LB[AR1, P#1.0];  // ..Store Byte 1
         L     #Pfister_BlkMove_Len;  // Load Packed length
         T     LW[AR1, P#2.0];  // ..Store byte 2/3
         L     0;  // used with DB else "0"
         T     LW[AR1, P#4.0];  // ..Store byte 4/5
         L     #Pfister_Offset;  // Source offset (Variable for Node's)
         SLD   3;  // with offset
         OD    16#8100_0000;  // Input Area (I/O) Code (S7)
         T     LD[AR1, P#6.0];  // ..Store byte 6/7/8/9

         LAR1;  // Load start point of cyclic data
         TAR1  #DummyDWord;  // Store in temp. point
         L     #DummyDWord;  // Load temp. point
         T     #Addr_InstanceDB;  // Store start point as DB address

         LAR1;  // Make AR1 point to calling program stack
         L     16#10;  // ANY Syntax ID
         T     LB[AR1, P#0.0];  // ..Store Byte 0
         L     16#02;  // Data Type = Byte
         T     LB[AR1, P#1.0];  // ..Store Byte 1
         L     #Pfister_BlkMove_Len;  // Load Packed length
         T     LW[AR1, P#2.0];  // ..Store Byte 2/3
         L     #BlockInfo.DB_Number;  // used with DB use No. else "0"
         T     LW[AR1, P#4.0];  // ..Store byte 4/5
         L     #Addr_InstanceDB;  // Load Instance DB Start address
         L     16#8500_0000;
         -D;
         L     16#8400_0000;
         +D;
         T     LD[AR1, P#6.0];  // ..Store byte 6/7/8/9
END_REGION

REGION Network 8: Read from Pfister Feeder
   #RET_VAL_Input := BLKMOV(SRCBLK := #IO_Pointer, DSTBLK => #DB_Pointer);
END_REGION

REGION Network 9: Check if WatchDog Counter has bee updated by Pfister
   #WatchDog_Same := #Rx.AdministrationNo = #Tx.AdministrationNo;
END_REGION

REGION Network 10
   "ACESYS_SecTimer_INT"(START := NOT #WatchDog_Same,
                         SEC := #Sec_Pulse,
                         PRE := 5,
                         Mem := #Watchdog_Mem,
                         ACC => #DummyInt,
                         DN => #WatchDog_Elapsed,
                         TT => #DummyBool);
END_REGION

REGION Network 11
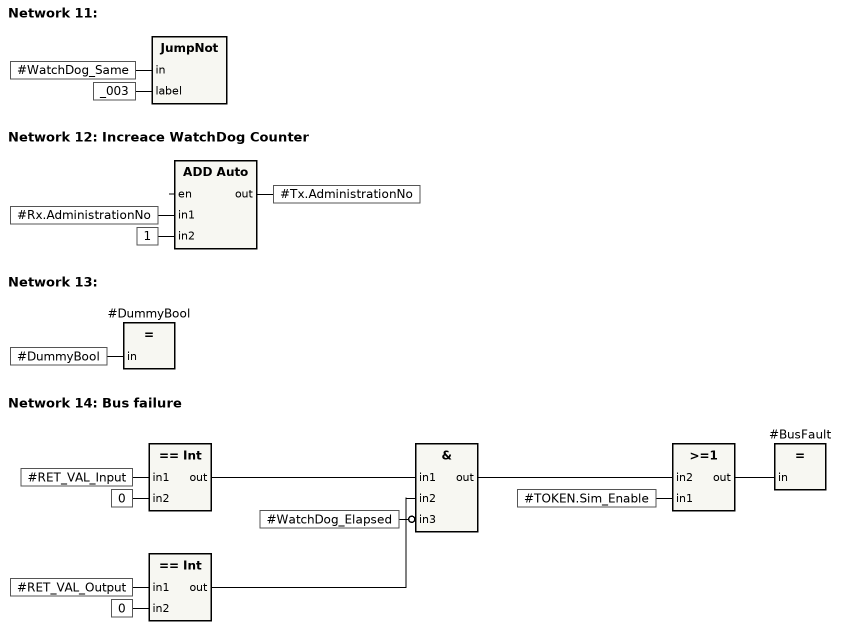
   // no SCL statement known for JumpNot: written as a call
   JumpNot(in := #WatchDog_Same, label := _003);
END_REGION

REGION Network 12: Increace WatchDog Counter
   #Tx.AdministrationNo := #Rx.AdministrationNo + 1;
END_REGION

REGION Network 13
   _003:
   #DummyBool := #DummyBool;
END_REGION

REGION Network 14: Bus failure
   // Build 002 - 26 March 2019 : Busfault bypassed during simulation
   #BusFault := ((#RET_VAL_Input = 0) AND (#RET_VAL_Output = 0) AND NOT #WatchDog_Elapsed) OR #TOKEN.Sim_Enable;
END_REGION

REGION Network 15: Config Optional values to be read
   // 1 - Feeder configuration
   //  2 - Prehopper configuration
   //  3 - Control value of feeder                  SY1 [rpm]
   //  4 - Present correction value                 QY1 [%]
   //  5 - Current of feeder                        II1 [A]
   //  6 - Loading at discharge                     WI1a [kg/r]
   //  7 - Relative loading at measuring            WI1 [%]
   //  8 - Setpoint of feed rate (feedback)         FY1 [t/h]
   //  9 - Totalizer 2                              FQ2 [t]
   // 10 - Loading residual quantity                QIL [t]
   // 11 - Setpoint loading quantity (feedback)     QYL [t]
   // 12 - Current of prefeeder                     II2 [A]
   // 13 - Dynamic setpoint of loading at infeed    WY1d [%]
   // 14 - Feed rate of prefeeder                   FI2 [t/h]
   // 15 - Setpoint of speed (position) of prefe.   SY2 [rpm] / GY2 [%]
   // 16 - Speed (position) of prefeeder            SI2 [rpm] / GI2 [%]
   // 17 - Current of refilling                     II3 [A]
   // 18 - Discharge capacity of refilling device   FI3 [t/h]
   // 19 - Accepted correction value                QY1a [%]
   // 20 - Nominal check quantity                   WY3 [t]
   // 
   // 
   // 21 - Present setpoint of level in prehopper   LY3 [t]
   // 22 - Pressure force                           PI3 [t]
   // 23 - Quantity fed by feeder                   FQ3 [t]
   // 24 - Remote correction (feedback)             QY1r [%]
   // 25 - Setpoint of speed (position ) of refill  SY3 [rpm] / GY3 [%]
   // 26 - Speed (position) of refilling system     SI3 [rpm] / GI3 [%]
   // 27 - Total zero correction                    ID 31.54[%]
   // 28 - Weighed quantity of prehopper            WI3 [t]
   // 29 - Level of material in silo                LI4 [t]
   // 30 - Reserve value 1RVr1
   // 31 - Reserve value 2RVr2
   // 32 - Reserve status
   // 33 - Firmware Version
   // 34 - Max Feed Rate                            FY1 max [t/h]
   // 35 - Weighing Range Prehopper                 [t]     
   // 
   // Build 008 - 24 April 2018 : Memory bit changed temp for TIA migration
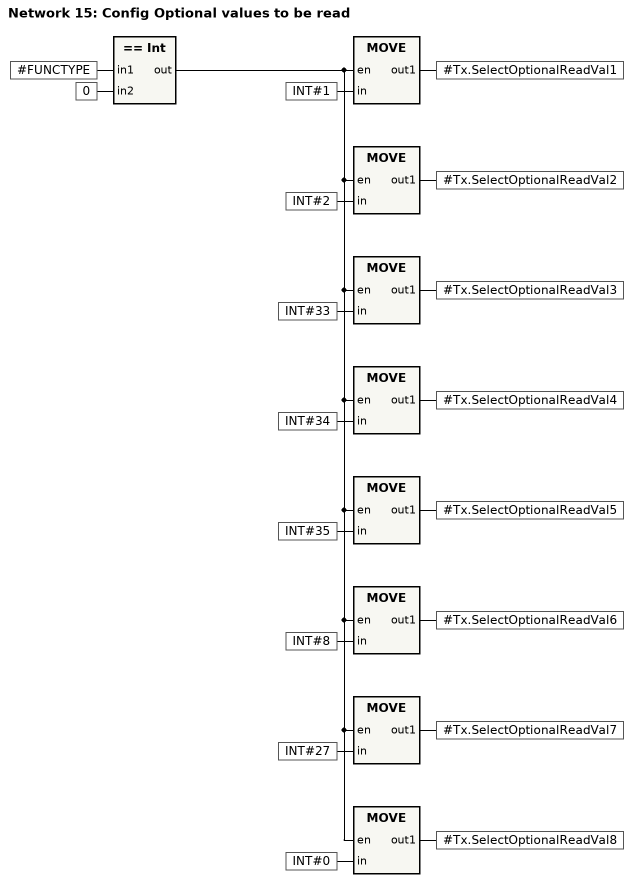
   IF #FUNCTYPE = 0 THEN
       #Tx.SelectOptionalReadVal1 := INT#1;
       #Tx.SelectOptionalReadVal2 := INT#2;
       #Tx.SelectOptionalReadVal3 := INT#33;
       #Tx.SelectOptionalReadVal4 := INT#34;
       #Tx.SelectOptionalReadVal5 := INT#35;
       #Tx.SelectOptionalReadVal6 := INT#8;
       #Tx.SelectOptionalReadVal7 := INT#27;
       #Tx.SelectOptionalReadVal8 := INT#0;
   END_IF;
END_REGION

REGION Network 16: GDC- Config Optional values to be read
   // Build 07 - 09 Jan 2022(VIV-IN) GDC Controller Function Type Added
   // 
   // GDC Controller Optinal Read Value
   // 
   // 19 - Feeder Configuration
   // 20 - Firmware
   // 21- Range Feed
   // 22 - Range Pre Hopper
   // 13 - Total OLC
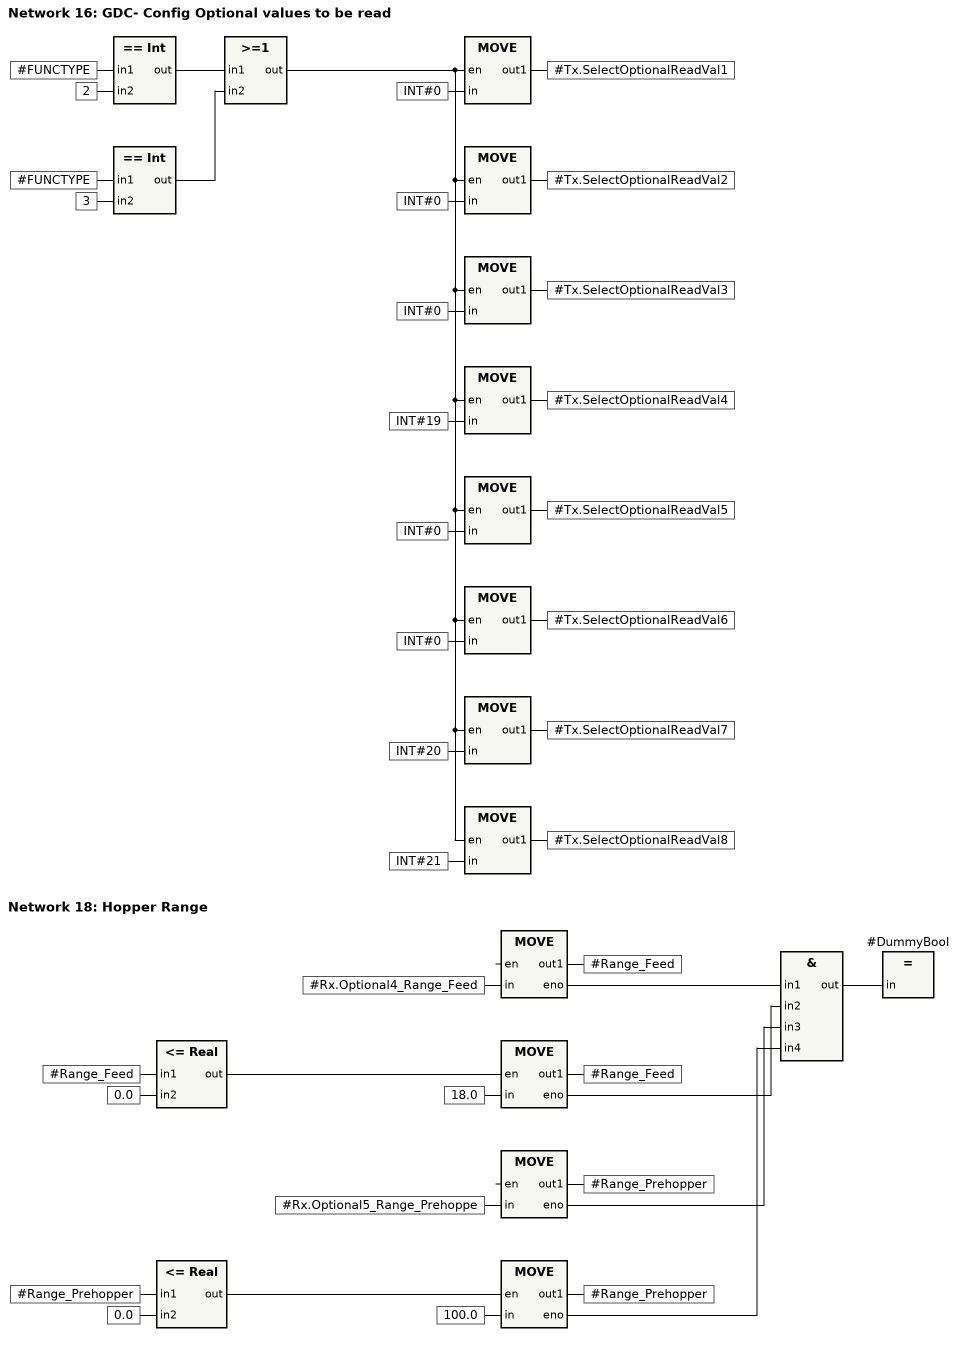
   IF (#FUNCTYPE = 2) OR (#FUNCTYPE = 3) THEN
       #Tx.SelectOptionalReadVal1 := INT#0;
       #Tx.SelectOptionalReadVal2 := INT#0;
       #Tx.SelectOptionalReadVal3 := INT#0;
       #Tx.SelectOptionalReadVal4 := INT#19;
       #Tx.SelectOptionalReadVal5 := INT#0;
       #Tx.SelectOptionalReadVal6 := INT#0;
       #Tx.SelectOptionalReadVal7 := INT#20;
       #Tx.SelectOptionalReadVal8 := INT#21;
   END_IF;
END_REGION

REGION Network 18: Hopper Range
   // ENO of a box is taken as its EN; it also drops when the box reports an error
   #Range_Feed := #Rx.Optional4_Range_Feed;
   #_w1 := #Range_Feed <= 0.0;
   IF #_w1 THEN #Range_Feed := 18.0; END_IF;
   #Range_Prehopper := #Rx.Optional5_Range_Prehoppe;
   #_w2 := #Range_Prehopper <= 0.0;
   IF #_w2 THEN #Range_Prehopper := 100.0; END_IF;
   #DummyBool := #_w1 AND #_w2;
END_REGION

REGION Network 19: Feeder Type
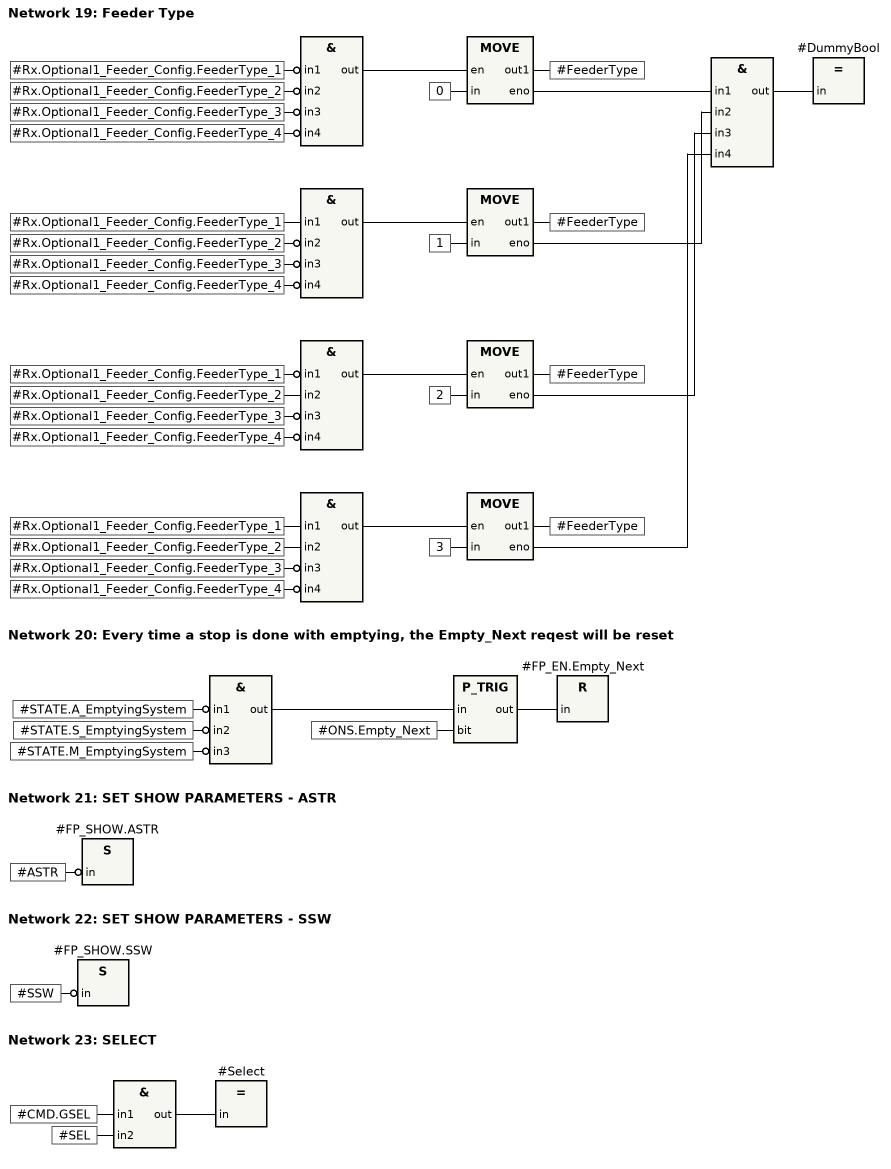
   // ENO of a box is taken as its EN; it also drops when the box reports an error
   #_w1 := NOT #Rx.Optional1_Feeder_Config.FeederType_1 AND NOT #Rx.Optional1_Feeder_Config.FeederType_2 AND NOT #Rx.Optional1_Feeder_Config.FeederType_3 AND NOT #Rx.Optional1_Feeder_Config.FeederType_4;
   IF #_w1 THEN #FeederType := 0; END_IF;
   #_w2 := #Rx.Optional1_Feeder_Config.FeederType_1 AND NOT #Rx.Optional1_Feeder_Config.FeederType_2 AND NOT #Rx.Optional1_Feeder_Config.FeederType_3 AND NOT #Rx.Optional1_Feeder_Config.FeederType_4;
   IF #_w2 THEN #FeederType := 1; END_IF;
   #_w3 := NOT #Rx.Optional1_Feeder_Config.FeederType_1 AND #Rx.Optional1_Feeder_Config.FeederType_2 AND NOT #Rx.Optional1_Feeder_Config.FeederType_3 AND NOT #Rx.Optional1_Feeder_Config.FeederType_4;
   IF #_w3 THEN #FeederType := 2; END_IF;
   #_w4 := #Rx.Optional1_Feeder_Config.FeederType_1 AND #Rx.Optional1_Feeder_Config.FeederType_2 AND NOT #Rx.Optional1_Feeder_Config.FeederType_3 AND NOT #Rx.Optional1_Feeder_Config.FeederType_4;
   IF #_w4 THEN #FeederType := 3; END_IF;
   #DummyBool := #_w1 AND #_w2 AND #_w3 AND #_w4;
END_REGION

REGION Network 20: Every time a stop is done with emptying, the Empty_Next reqest will be reset
   #_w1 := NOT #STATE.A_EmptyingSystem AND NOT #STATE.S_EmptyingSystem AND NOT #STATE.M_EmptyingSystem;
   #_w2 := #_w1 AND NOT #ONS.Empty_Next;   // rising edge
   #ONS.Empty_Next := #_w1;
   IF #_w2 THEN #FP_EN.Empty_Next := FALSE; END_IF;
END_REGION

REGION Network 21: SET SHOW PARAMETERS - ASTR
   IF NOT #ASTR THEN #FP_SHOW.ASTR := TRUE; END_IF;
END_REGION

REGION Network 22: SET SHOW PARAMETERS - SSW
   IF NOT #SSW THEN #FP_SHOW.SSW := TRUE; END_IF;
END_REGION

REGION Network 23: SELECT
   #Select := #CMD.GSEL AND #SEL;
END_REGION

REGION Network 24: INIT MODES FOR THIS UNIT
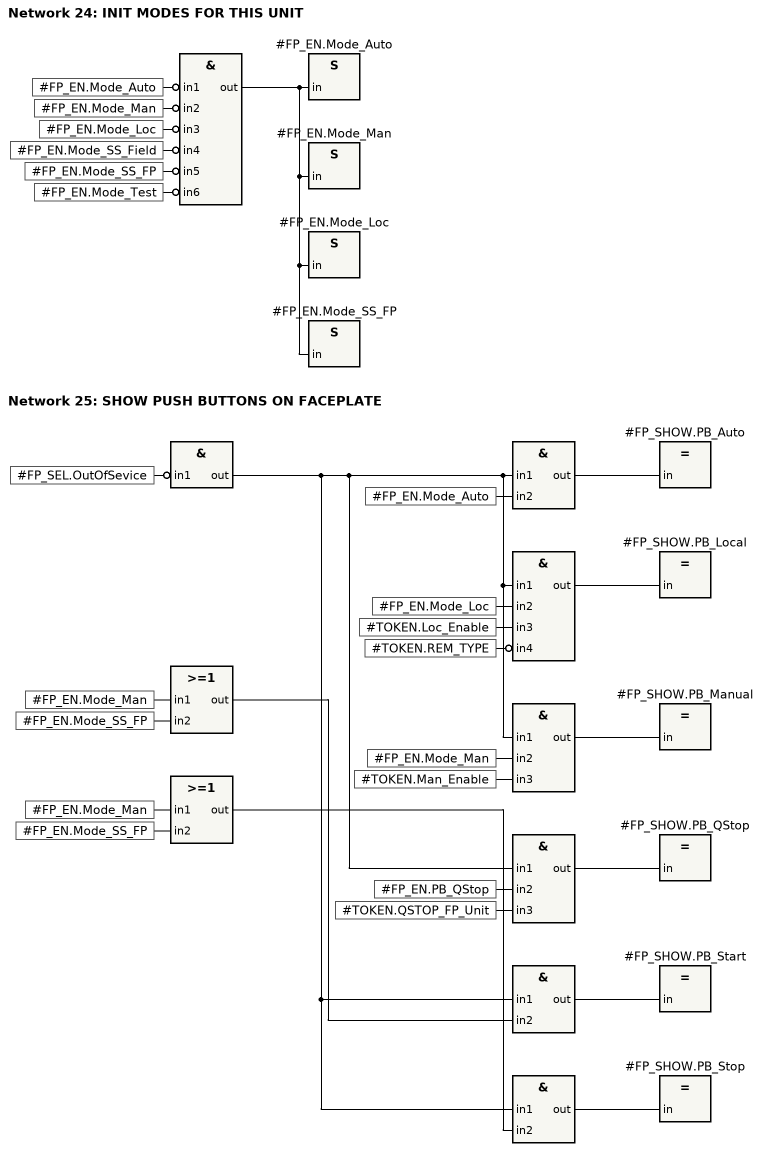
   #_w1 := NOT #FP_EN.Mode_Auto AND NOT #FP_EN.Mode_Man AND NOT #FP_EN.Mode_Loc AND NOT #FP_EN.Mode_SS_Field AND NOT #FP_EN.Mode_SS_FP AND NOT #FP_EN.Mode_Test;
   IF #_w1 THEN
       #FP_EN.Mode_Auto := TRUE;
       #FP_EN.Mode_Man := TRUE;
       #FP_EN.Mode_Loc := TRUE;
       #FP_EN.Mode_SS_FP := TRUE;
   END_IF;
END_REGION

REGION Network 25: SHOW PUSH BUTTONS ON FACEPLATE
   // Build 002 - 26 March 2019 : Loc_type flag removed from Show_PB_local
   #FP_SHOW.PB_Auto := NOT #FP_SEL.OutOfSevice AND #FP_EN.Mode_Auto;
   #FP_SHOW.PB_Local := NOT #FP_SEL.OutOfSevice AND #FP_EN.Mode_Loc AND #TOKEN.Loc_Enable AND NOT #TOKEN.REM_TYPE;
   #FP_SHOW.PB_Manual := NOT #FP_SEL.OutOfSevice AND #FP_EN.Mode_Man AND #TOKEN.Man_Enable;
   #FP_SHOW.PB_QStop := NOT #FP_SEL.OutOfSevice AND #FP_EN.PB_QStop AND #TOKEN.QSTOP_FP_Unit;
   #FP_SHOW.PB_Start := NOT #FP_SEL.OutOfSevice AND (#FP_EN.Mode_Man OR #FP_EN.Mode_SS_FP);
   #FP_SHOW.PB_Stop := NOT #FP_SEL.OutOfSevice AND (#FP_EN.Mode_Man OR #FP_EN.Mode_SS_FP);
END_REGION

REGION Network 26: DIMOUT BUTTONS ON FACEPLATE - Auto
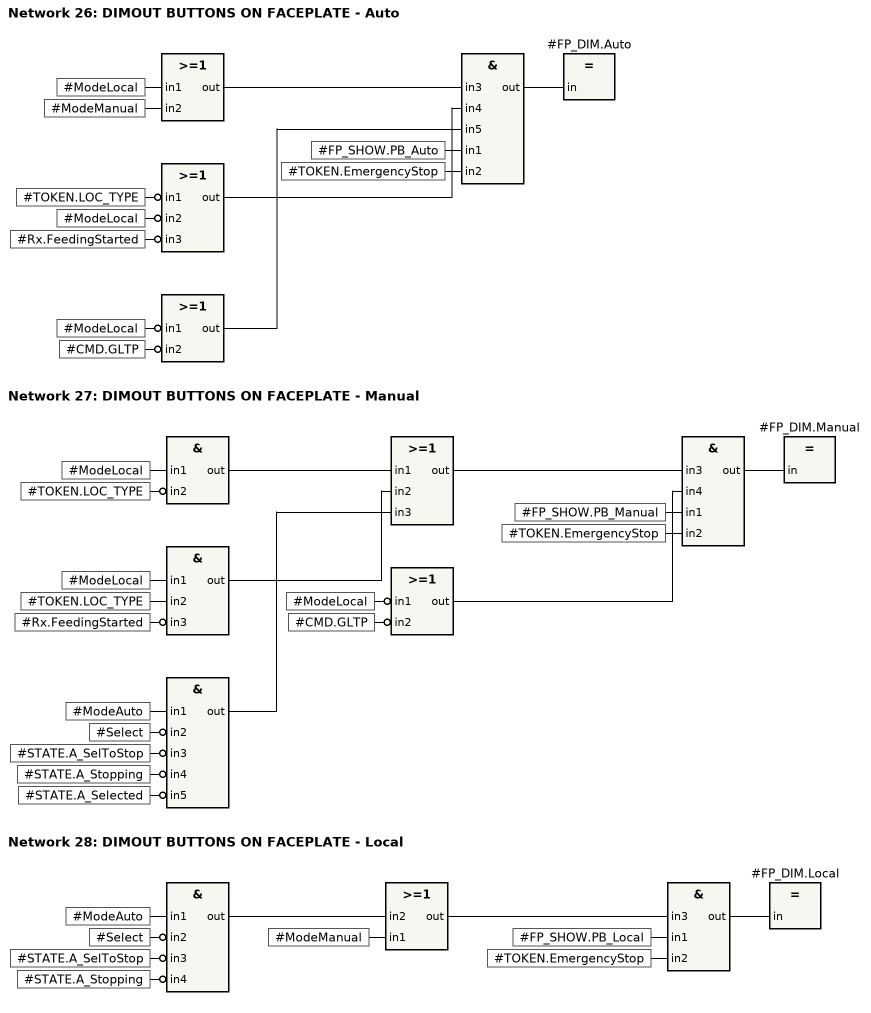
   #FP_DIM.Auto := (#ModeLocal OR #ModeManual) AND (NOT #TOKEN.LOC_TYPE OR NOT #ModeLocal OR NOT #Rx.FeedingStarted) AND (NOT #ModeLocal OR NOT #CMD.GLTP) AND #FP_SHOW.PB_Auto AND #TOKEN.EmergencyStop;
END_REGION

REGION Network 27: DIMOUT BUTTONS ON FACEPLATE - Manual
   #FP_DIM.Manual := ((#ModeLocal AND NOT #TOKEN.LOC_TYPE) OR (#ModeLocal AND #TOKEN.LOC_TYPE AND NOT #Rx.FeedingStarted) OR (#ModeAuto AND NOT #Select AND NOT #STATE.A_SelToStop AND NOT #STATE.A_Stopping AND NOT #STATE.A_Selected)) AND (NOT #ModeLocal OR NOT #CMD.GLTP) AND #FP_SHOW.PB_Manual AND #TOKEN.EmergencyStop;
END_REGION

REGION Network 28: DIMOUT BUTTONS ON FACEPLATE - Local
   #FP_DIM.Local := ((#ModeAuto AND NOT #Select AND NOT #STATE.A_SelToStop AND NOT #STATE.A_Stopping) OR #ModeManual) AND #FP_SHOW.PB_Local AND #TOKEN.EmergencyStop;
END_REGION

REGION Network 29: DIMOUT BUTTONS ON FACEPLATE - Stop
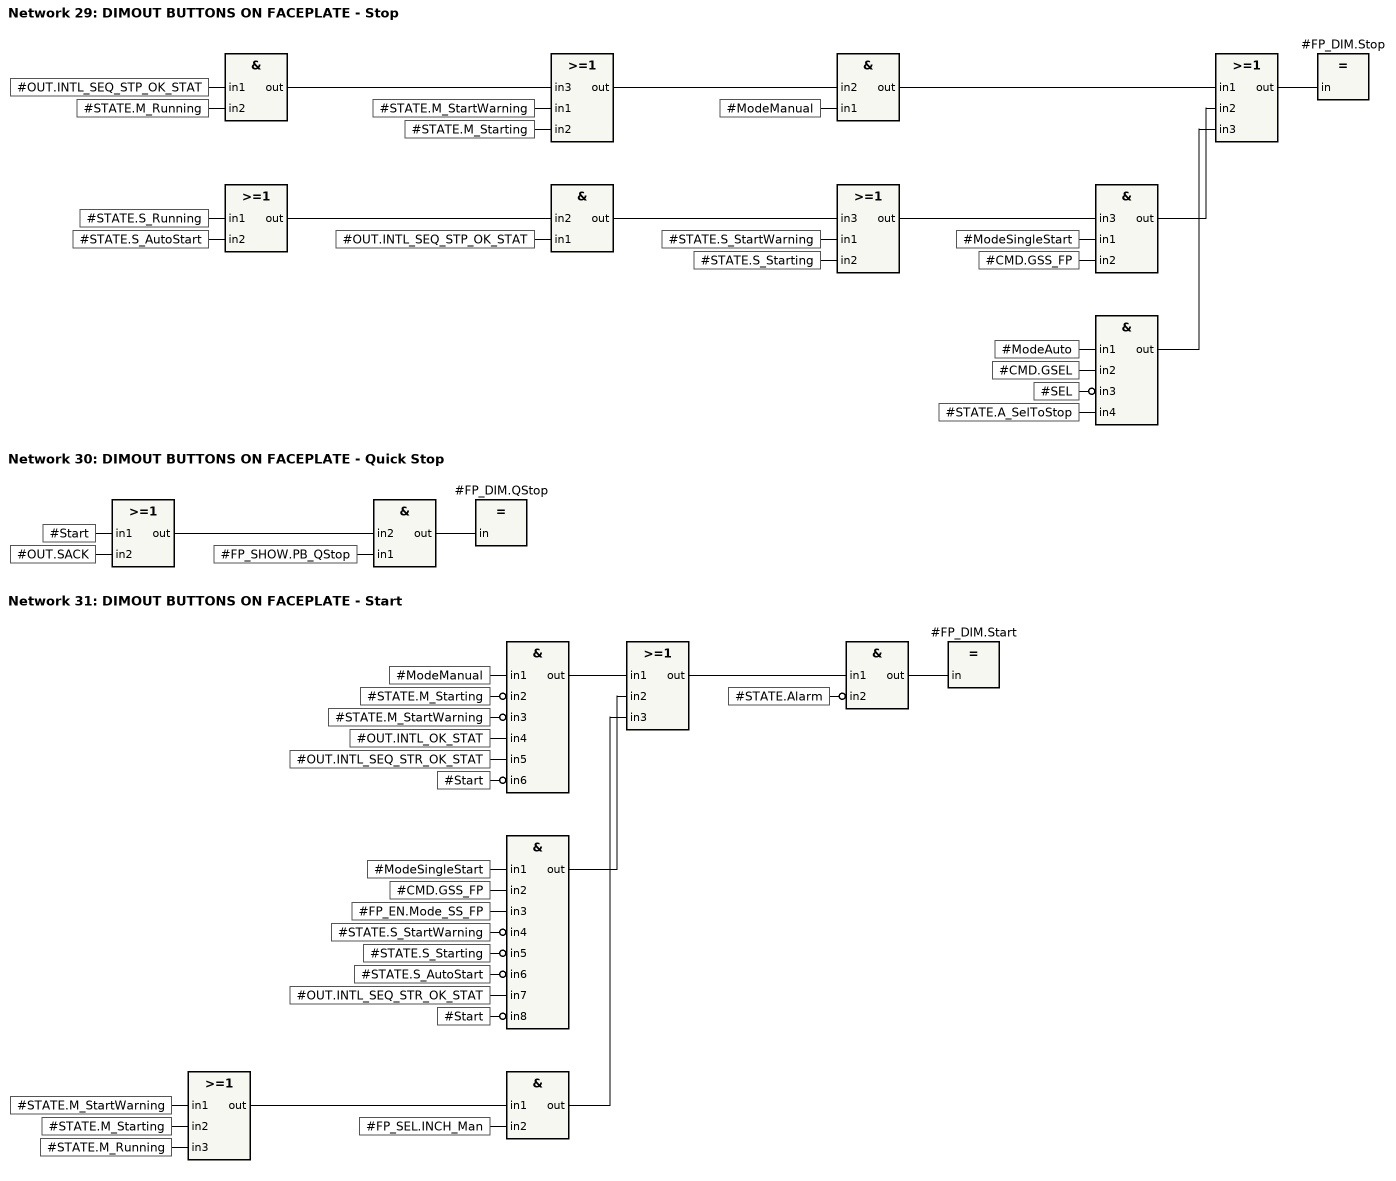
   #FP_DIM.Stop := (((#OUT.INTL_SEQ_STP_OK_STAT AND #STATE.M_Running) OR #STATE.M_StartWarning OR #STATE.M_Starting) AND #ModeManual) OR ((((#STATE.S_Running OR #STATE.S_AutoStart) AND #OUT.INTL_SEQ_STP_OK_STAT) OR #STATE.S_StartWarning OR #STATE.S_Starting) AND #ModeSingleStart AND #CMD.GSS_FP) OR (#ModeAuto AND #CMD.GSEL AND NOT #SEL AND #STATE.A_SelToStop);
END_REGION

REGION Network 30: DIMOUT BUTTONS ON FACEPLATE - Quick Stop
   #FP_DIM.QStop := (#Start OR #OUT.SACK) AND #FP_SHOW.PB_QStop;
END_REGION

REGION Network 31: DIMOUT BUTTONS ON FACEPLATE - Start
   #FP_DIM.Start := ((#ModeManual AND NOT #STATE.M_Starting AND NOT #STATE.M_StartWarning AND #OUT.INTL_OK_STAT AND #OUT.INTL_SEQ_STR_OK_STAT AND NOT #Start) OR (#ModeSingleStart AND #CMD.GSS_FP AND #FP_EN.Mode_SS_FP AND NOT #STATE.S_StartWarning AND NOT #STATE.S_Starting AND NOT #STATE.S_AutoStart AND #OUT.INTL_SEQ_STR_OK_STAT AND NOT #Start) OR ((#STATE.M_StartWarning OR #STATE.M_Starting OR #STATE.M_Running) AND #FP_SEL.INCH_Man)) AND NOT #STATE.Alarm;
END_REGION

REGION Network 32: MODE Handling - Auto Mode
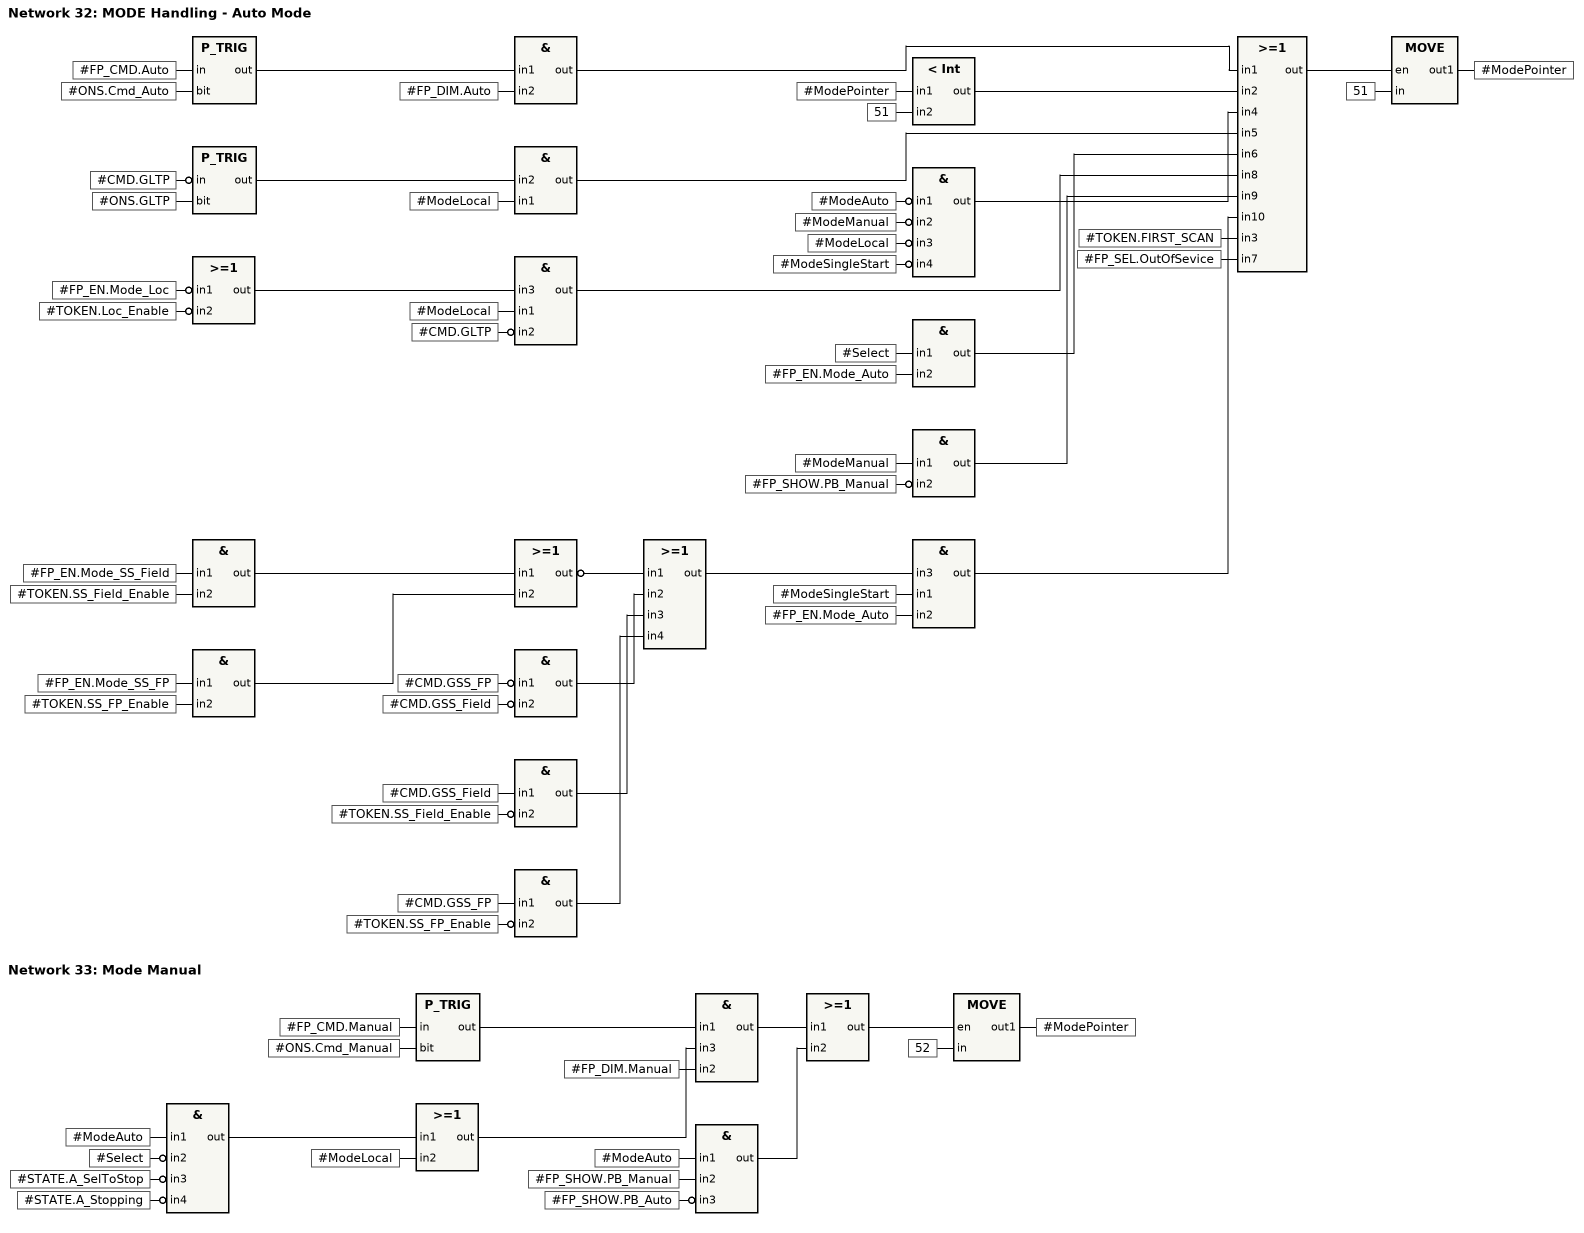
   #_w1 := #FP_CMD.Auto AND NOT #ONS.Cmd_Auto;   // rising edge
   #ONS.Cmd_Auto := #FP_CMD.Auto;
   #_w2 := NOT #CMD.GLTP AND NOT #ONS.GLTP;   // rising edge
   #ONS.GLTP := NOT #CMD.GLTP;
   IF (#_w1 AND #FP_DIM.Auto) OR (#ModePointer < 51) OR (NOT #ModeAuto AND NOT #ModeManual AND NOT #ModeLocal AND NOT #ModeSingleStart) OR (#_w2 AND #ModeLocal) OR (#Select AND #FP_EN.Mode_Auto) OR ((NOT #FP_EN.Mode_Loc OR NOT #TOKEN.Loc_Enable) AND #ModeLocal AND NOT #CMD.GLTP) OR (#ModeManual AND NOT #FP_SHOW.PB_Manual) OR ((NOT ((#FP_EN.Mode_SS_Field AND #TOKEN.SS_Field_Enable) OR (#FP_EN.Mode_SS_FP AND #TOKEN.SS_FP_Enable)) OR (NOT #CMD.GSS_FP AND NOT #CMD.GSS_Field) OR (#CMD.GSS_Field AND NOT #TOKEN.SS_Field_Enable) OR (#CMD.GSS_FP AND NOT #TOKEN.SS_FP_Enable)) AND #ModeSingleStart AND #FP_EN.Mode_Auto) OR #TOKEN.FIRST_SCAN OR #FP_SEL.OutOfSevice THEN
       #ModePointer := 51;
   END_IF;
END_REGION

REGION Network 33: Mode Manual
   #_w1 := #FP_CMD.Manual AND NOT #ONS.Cmd_Manual;   // rising edge
   #ONS.Cmd_Manual := #FP_CMD.Manual;
   IF (#_w1 AND ((#ModeAuto AND NOT #Select AND NOT #STATE.A_SelToStop AND NOT #STATE.A_Stopping) OR #ModeLocal) AND #FP_DIM.Manual) OR (#ModeAuto AND #FP_SHOW.PB_Manual AND NOT #FP_SHOW.PB_Auto) THEN
       #ModePointer := 52;
   END_IF;
END_REGION

REGION Network 34: Mode Single Start
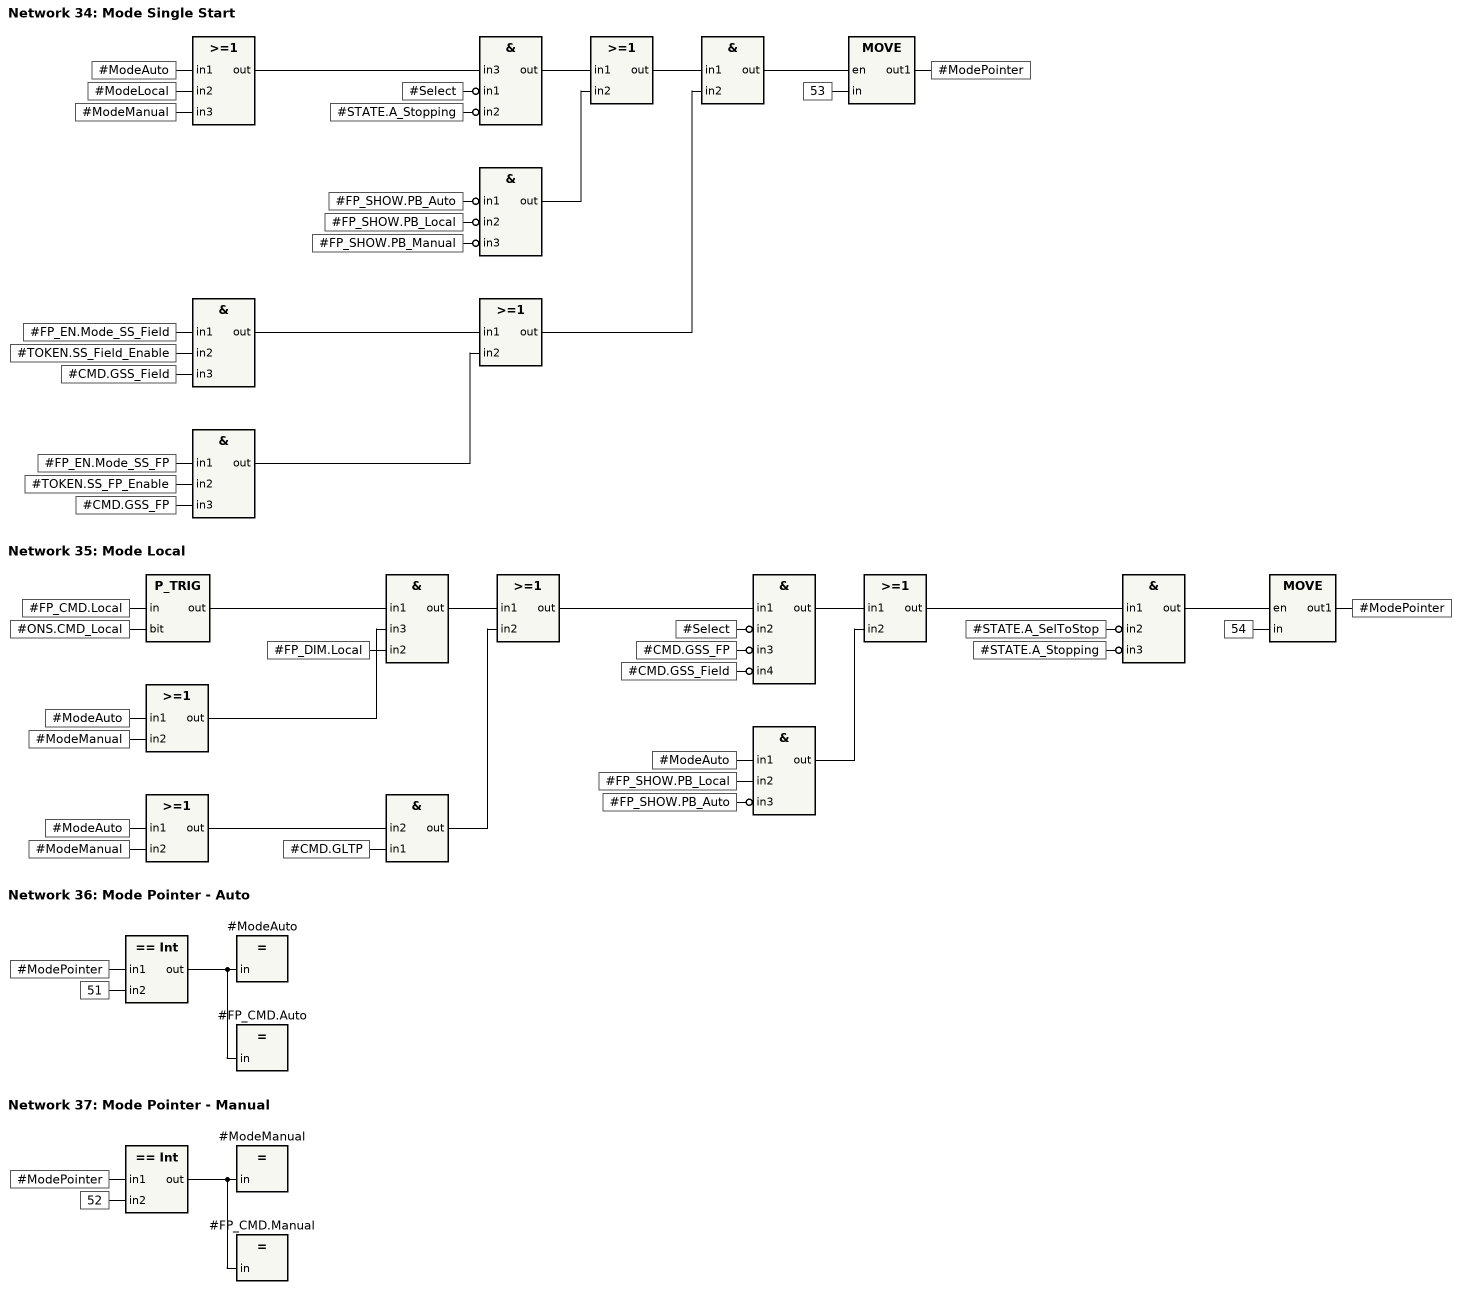
   IF (((#ModeAuto OR #ModeLocal OR #ModeManual) AND NOT #Select AND NOT #STATE.A_Stopping) OR (NOT #FP_SHOW.PB_Auto AND NOT #FP_SHOW.PB_Local AND NOT #FP_SHOW.PB_Manual)) AND ((#FP_EN.Mode_SS_Field AND #TOKEN.SS_Field_Enable AND #CMD.GSS_Field) OR (#FP_EN.Mode_SS_FP AND #TOKEN.SS_FP_Enable AND #CMD.GSS_FP)) THEN
       #ModePointer := 53;
   END_IF;
END_REGION

REGION Network 35: Mode Local
   #_w1 := #FP_CMD.Local AND NOT #ONS.CMD_Local;   // rising edge
   #ONS.CMD_Local := #FP_CMD.Local;
   IF ((((#_w1 AND (#ModeAuto OR #ModeManual) AND #FP_DIM.Local) OR ((#ModeAuto OR #ModeManual) AND #CMD.GLTP)) AND NOT #Select AND NOT #CMD.GSS_FP AND NOT #CMD.GSS_Field) OR (#ModeAuto AND #FP_SHOW.PB_Local AND NOT #FP_SHOW.PB_Auto)) AND NOT #STATE.A_SelToStop AND NOT #STATE.A_Stopping THEN
       #ModePointer := 54;
   END_IF;
END_REGION

REGION Network 36: Mode Pointer - Auto
   #ModeAuto := #ModePointer = 51;
   #FP_CMD.Auto := #ModeAuto;
END_REGION

REGION Network 37: Mode Pointer - Manual
   #ModeManual := #ModePointer = 52;
   #FP_CMD.Manual := #ModeManual;
END_REGION

REGION Network 38: Mode Pointer - SS
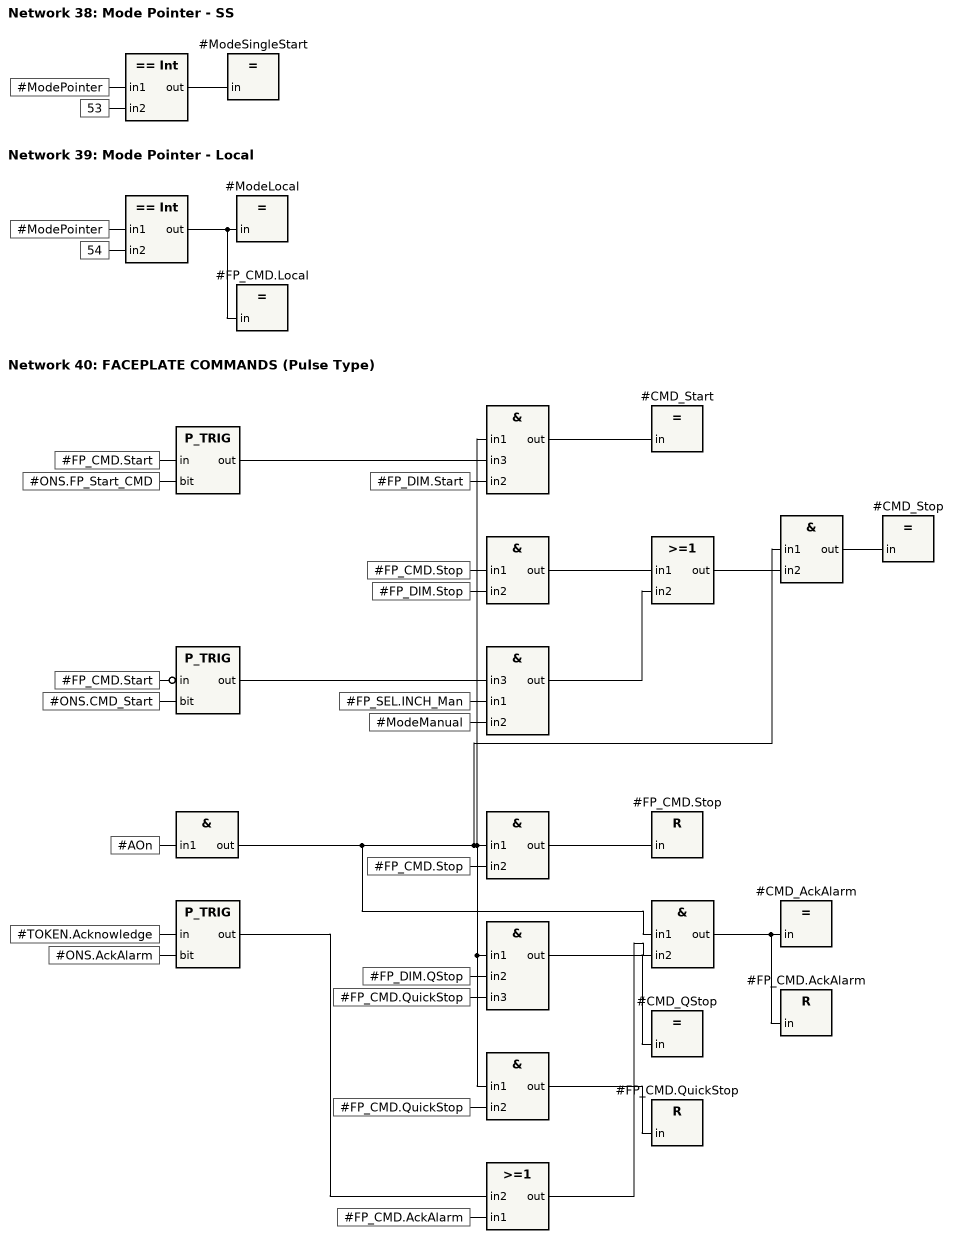
   #ModeSingleStart := #ModePointer = 53;
END_REGION

REGION Network 39: Mode Pointer - Local
   #ModeLocal := #ModePointer = 54;
   #FP_CMD.Local := #ModeLocal;
END_REGION

REGION Network 40: FACEPLATE COMMANDS (Pulse Type)
   #_w1 := #FP_CMD.Start AND NOT #ONS.FP_Start_CMD;   // rising edge
   #ONS.FP_Start_CMD := #FP_CMD.Start;
   #CMD_Start := #AOn AND #_w1 AND #FP_DIM.Start;
   #_w2 := NOT #FP_CMD.Start AND NOT #ONS.CMD_Start;   // rising edge
   #ONS.CMD_Start := NOT #FP_CMD.Start;
   #CMD_Stop := #AOn AND ((#FP_CMD.Stop AND #FP_DIM.Stop) OR (#_w2 AND #FP_SEL.INCH_Man AND #ModeManual));
   IF #AOn AND #FP_CMD.Stop THEN #FP_CMD.Stop := FALSE; END_IF;
   #CMD_QStop := #AOn AND #FP_DIM.QStop AND #FP_CMD.QuickStop;
   IF #AOn AND #FP_CMD.QuickStop THEN #FP_CMD.QuickStop := FALSE; END_IF;
   #_w3 := #TOKEN.Acknowledge AND NOT #ONS.AckAlarm;   // rising edge
   #ONS.AckAlarm := #TOKEN.Acknowledge;
   #CMD_AckAlarm := #AOn AND (#_w3 OR #FP_CMD.AckAlarm);
   IF #CMD_AckAlarm THEN #FP_CMD.AckAlarm := FALSE; END_IF;
END_REGION

REGION Network 41
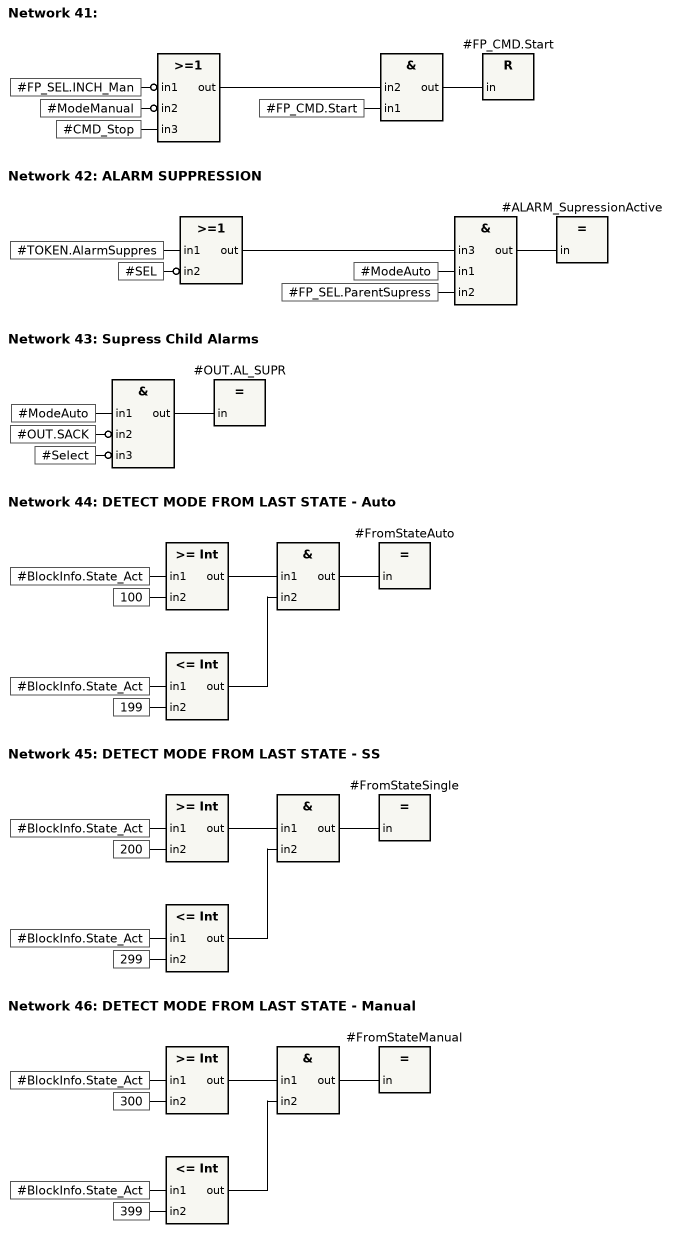
   IF (NOT #FP_SEL.INCH_Man OR NOT #ModeManual OR #CMD_Stop) AND #FP_CMD.Start THEN
       #FP_CMD.Start := FALSE;
   END_IF;
END_REGION

REGION Network 42: ALARM SUPPRESSION
   #ALARM_SupressionActive := (#TOKEN.AlarmSuppres OR NOT #SEL) AND #ModeAuto AND #FP_SEL.ParentSupress;
END_REGION

REGION Network 43: Supress Child Alarms
   #OUT.AL_SUPR := #ModeAuto AND NOT #OUT.SACK AND NOT #Select;
END_REGION

REGION Network 44: DETECT MODE FROM LAST STATE - Auto
   #FromStateAuto := (#BlockInfo.State_Act >= 100) AND (#BlockInfo.State_Act <= 199);
END_REGION

REGION Network 45: DETECT MODE FROM LAST STATE - SS
   #FromStateSingle := (#BlockInfo.State_Act >= 200) AND (#BlockInfo.State_Act <= 299);
END_REGION

REGION Network 46: DETECT MODE FROM LAST STATE - Manual
   #FromStateManual := (#BlockInfo.State_Act >= 300) AND (#BlockInfo.State_Act <= 399);
END_REGION

REGION Network 47: DETECT MODE FROM LAST STATE - Local
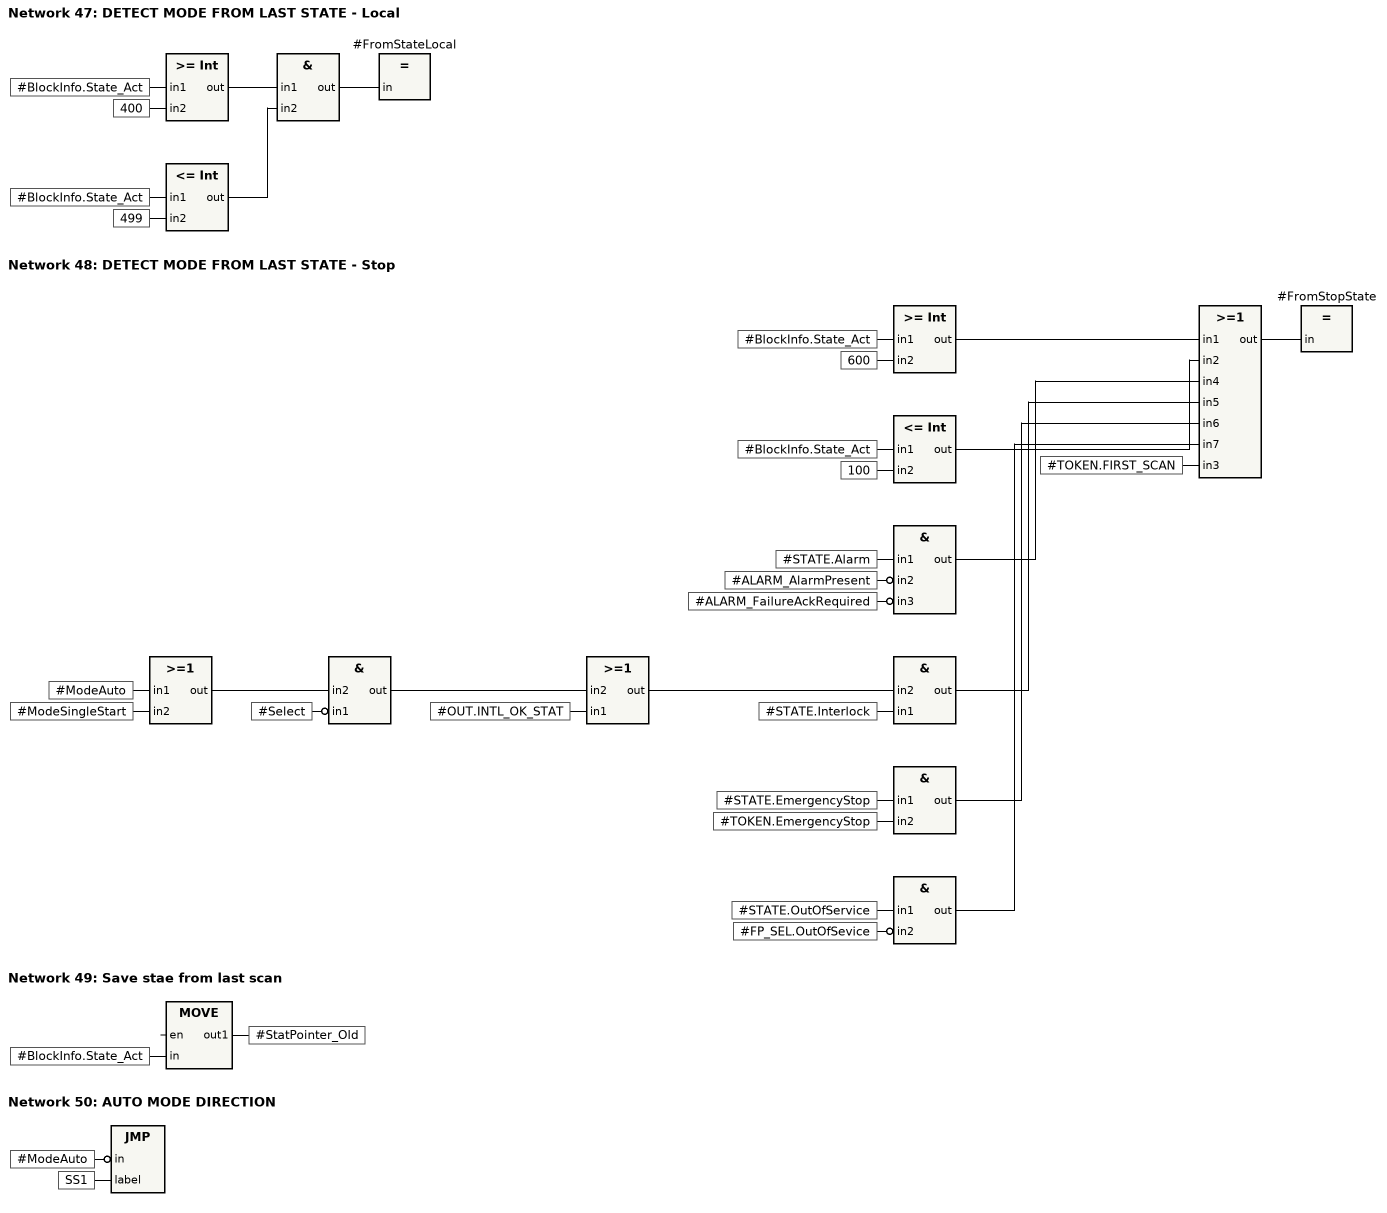
   #FromStateLocal := (#BlockInfo.State_Act >= 400) AND (#BlockInfo.State_Act <= 499);
END_REGION

REGION Network 48: DETECT MODE FROM LAST STATE - Stop
   #FromStopState := (#BlockInfo.State_Act >= 600) OR (#BlockInfo.State_Act <= 100) OR (#STATE.Alarm AND NOT #ALARM_AlarmPresent AND NOT #ALARM_FailureAckRequired) OR ((((#ModeAuto OR #ModeSingleStart) AND NOT #Select) OR #OUT.INTL_OK_STAT) AND #STATE.Interlock) OR (#STATE.EmergencyStop AND #TOKEN.EmergencyStop) OR (#STATE.OutOfService AND NOT #FP_SEL.OutOfSevice) OR #TOKEN.FIRST_SCAN;
END_REGION

REGION Network 49: Save stae from last scan
   #StatPointer_Old := #BlockInfo.State_Act;
END_REGION

REGION Network 50: AUTO MODE DIRECTION
   IF NOT #ModeAuto THEN GOTO SS1; END_IF;
END_REGION

REGION Network 51: State: Auto - Stopped
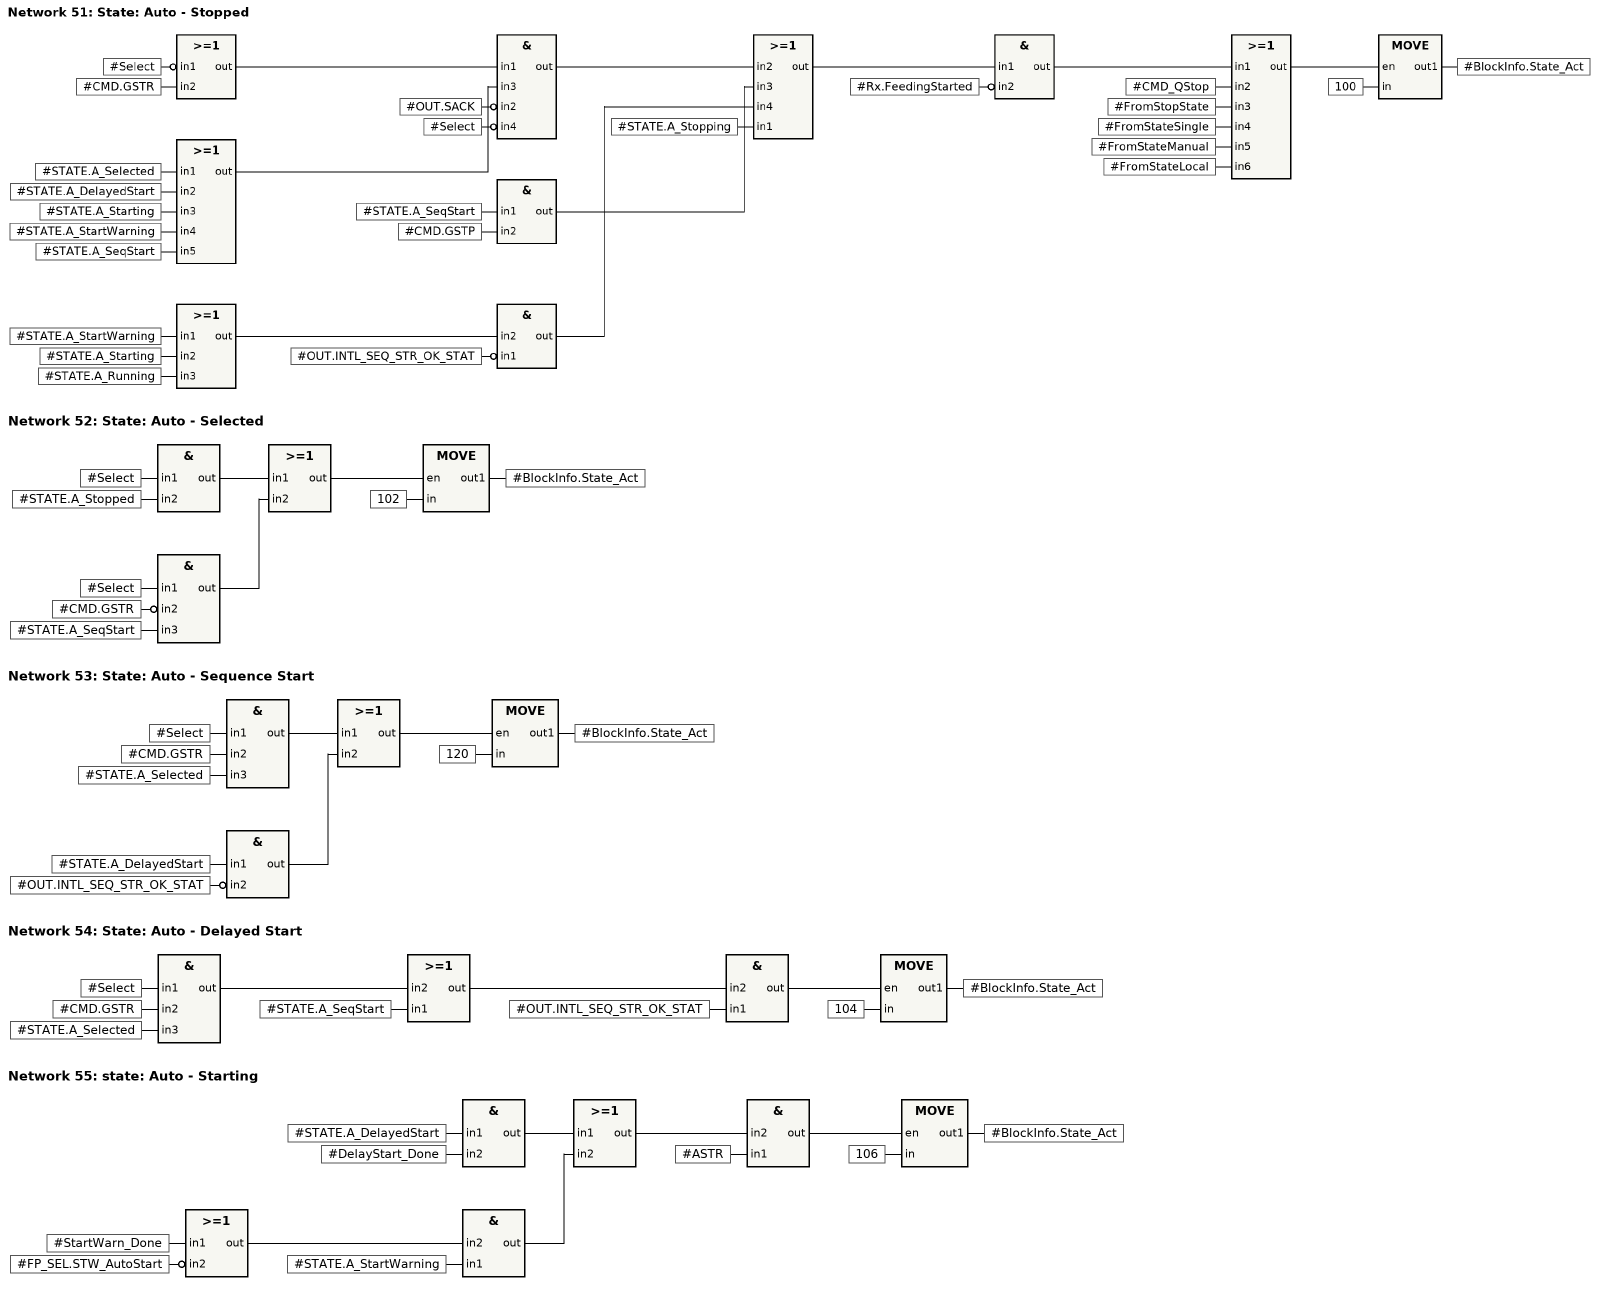
   IF ((((NOT #Select OR #CMD.GSTR) AND (#STATE.A_Selected OR #STATE.A_DelayedStart OR #STATE.A_Starting OR #STATE.A_StartWarning OR #STATE.A_SeqStart) AND NOT #OUT.SACK AND NOT #Select) OR (#STATE.A_SeqStart AND #CMD.GSTP) OR ((#STATE.A_StartWarning OR #STATE.A_Starting OR #STATE.A_Running) AND NOT #OUT.INTL_SEQ_STR_OK_STAT) OR #STATE.A_Stopping) AND NOT #Rx.FeedingStarted) OR #CMD_QStop OR #FromStopState OR #FromStateSingle OR #FromStateManual OR #FromStateLocal THEN
       #BlockInfo.State_Act := 100;
   END_IF;
END_REGION

REGION Network 52: State: Auto - Selected
   IF (#Select AND #STATE.A_Stopped) OR (#Select AND NOT #CMD.GSTR AND #STATE.A_SeqStart) THEN
       #BlockInfo.State_Act := 102;
   END_IF;
END_REGION

REGION Network 53: State: Auto - Sequence Start
   IF (#Select AND #CMD.GSTR AND #STATE.A_Selected) OR (#STATE.A_DelayedStart AND NOT #OUT.INTL_SEQ_STR_OK_STAT) THEN
       #BlockInfo.State_Act := 120;
   END_IF;
END_REGION

REGION Network 54: State: Auto - Delayed Start
   IF ((#Select AND #CMD.GSTR AND #STATE.A_Selected) OR #STATE.A_SeqStart) AND #OUT.INTL_SEQ_STR_OK_STAT THEN
       #BlockInfo.State_Act := 104;
   END_IF;
END_REGION

REGION Network 55: state: Auto - Starting
   IF ((#STATE.A_DelayedStart AND #DelayStart_Done) OR ((#StartWarn_Done OR NOT #FP_SEL.STW_AutoStart) AND #STATE.A_StartWarning)) AND #ASTR THEN
       #BlockInfo.State_Act := 106;
   END_IF;
END_REGION

REGION Network 56: State: Auto - Running
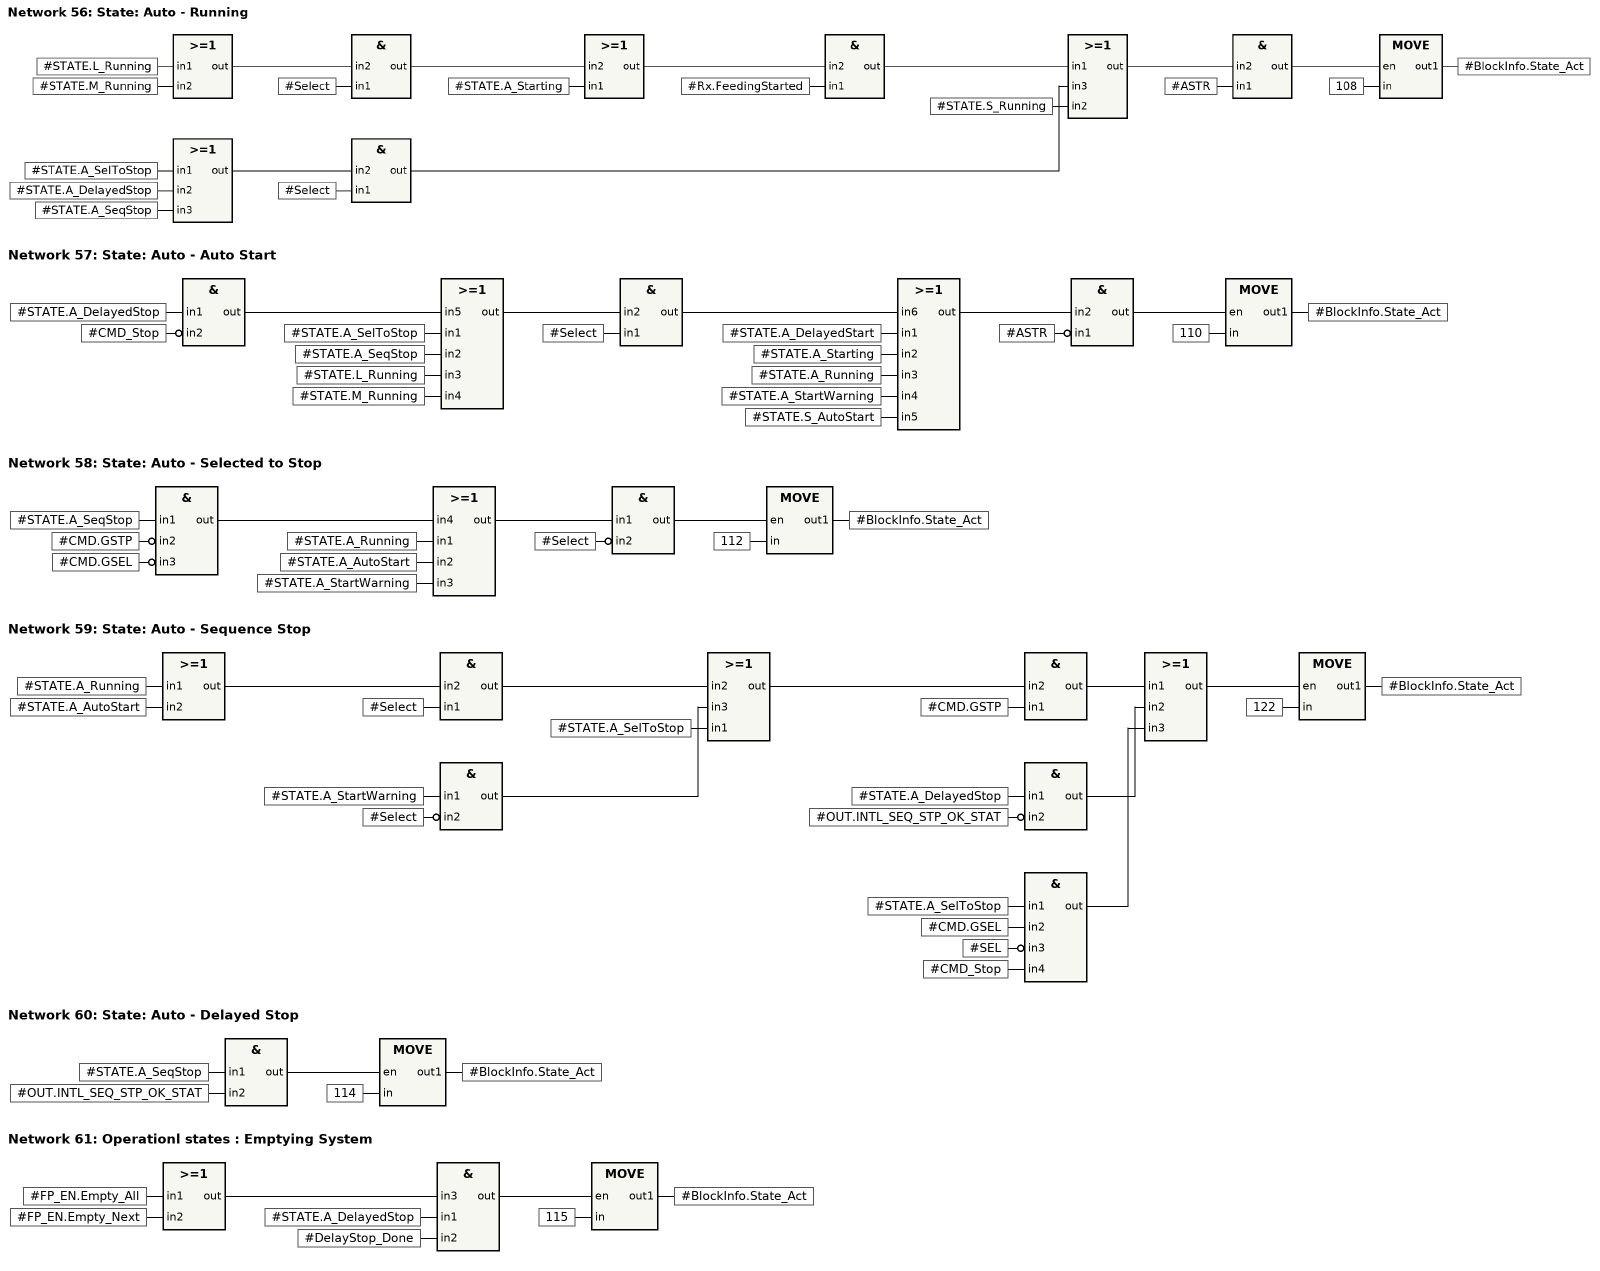
   IF (((((#STATE.L_Running OR #STATE.M_Running) AND #Select) OR #STATE.A_Starting) AND #Rx.FeedingStarted) OR ((#STATE.A_SelToStop OR #STATE.A_DelayedStop OR #STATE.A_SeqStop) AND #Select) OR #STATE.S_Running) AND #ASTR THEN
       #BlockInfo.State_Act := 108;
   END_IF;
END_REGION

REGION Network 57: State: Auto - Auto Start
   IF ((((#STATE.A_DelayedStop AND NOT #CMD_Stop) OR #STATE.A_SelToStop OR #STATE.A_SeqStop OR #STATE.L_Running OR #STATE.M_Running) AND #Select) OR #STATE.A_DelayedStart OR #STATE.A_Starting OR #STATE.A_Running OR #STATE.A_StartWarning OR #STATE.S_AutoStart) AND NOT #ASTR THEN
       #BlockInfo.State_Act := 110;
   END_IF;
END_REGION

REGION Network 58: State: Auto - Selected to Stop
   // Build 003 - 11 Jul 2019 (EXTBOB) : GSEL added to A_SeqStop with GSTP condition to move to Selected to Stop state from Seq stop state if group stop timer completes
   IF ((#STATE.A_SeqStop AND NOT #CMD.GSTP AND NOT #CMD.GSEL) OR #STATE.A_Running OR #STATE.A_AutoStart OR #STATE.A_StartWarning) AND NOT #Select THEN
       #BlockInfo.State_Act := 112;
   END_IF;
END_REGION

REGION Network 59: State: Auto - Sequence Stop
   IF ((((#STATE.A_Running OR #STATE.A_AutoStart) AND #Select) OR (#STATE.A_StartWarning AND NOT #Select) OR #STATE.A_SelToStop) AND #CMD.GSTP) OR (#STATE.A_DelayedStop AND NOT #OUT.INTL_SEQ_STP_OK_STAT) OR (#STATE.A_SelToStop AND #CMD.GSEL AND NOT #SEL AND #CMD_Stop) THEN
       #BlockInfo.State_Act := 122;
   END_IF;
END_REGION

REGION Network 60: State: Auto - Delayed Stop
   IF #STATE.A_SeqStop AND #OUT.INTL_SEQ_STP_OK_STAT THEN #BlockInfo.State_Act := 114; END_IF;
END_REGION

REGION Network 61: Operationl states : Emptying System
   IF (#FP_EN.Empty_All OR #FP_EN.Empty_Next) AND #STATE.A_DelayedStop AND #DelayStop_Done THEN
       #BlockInfo.State_Act := 115;
   END_IF;
END_REGION

REGION Network 62: State: Auto Stopping
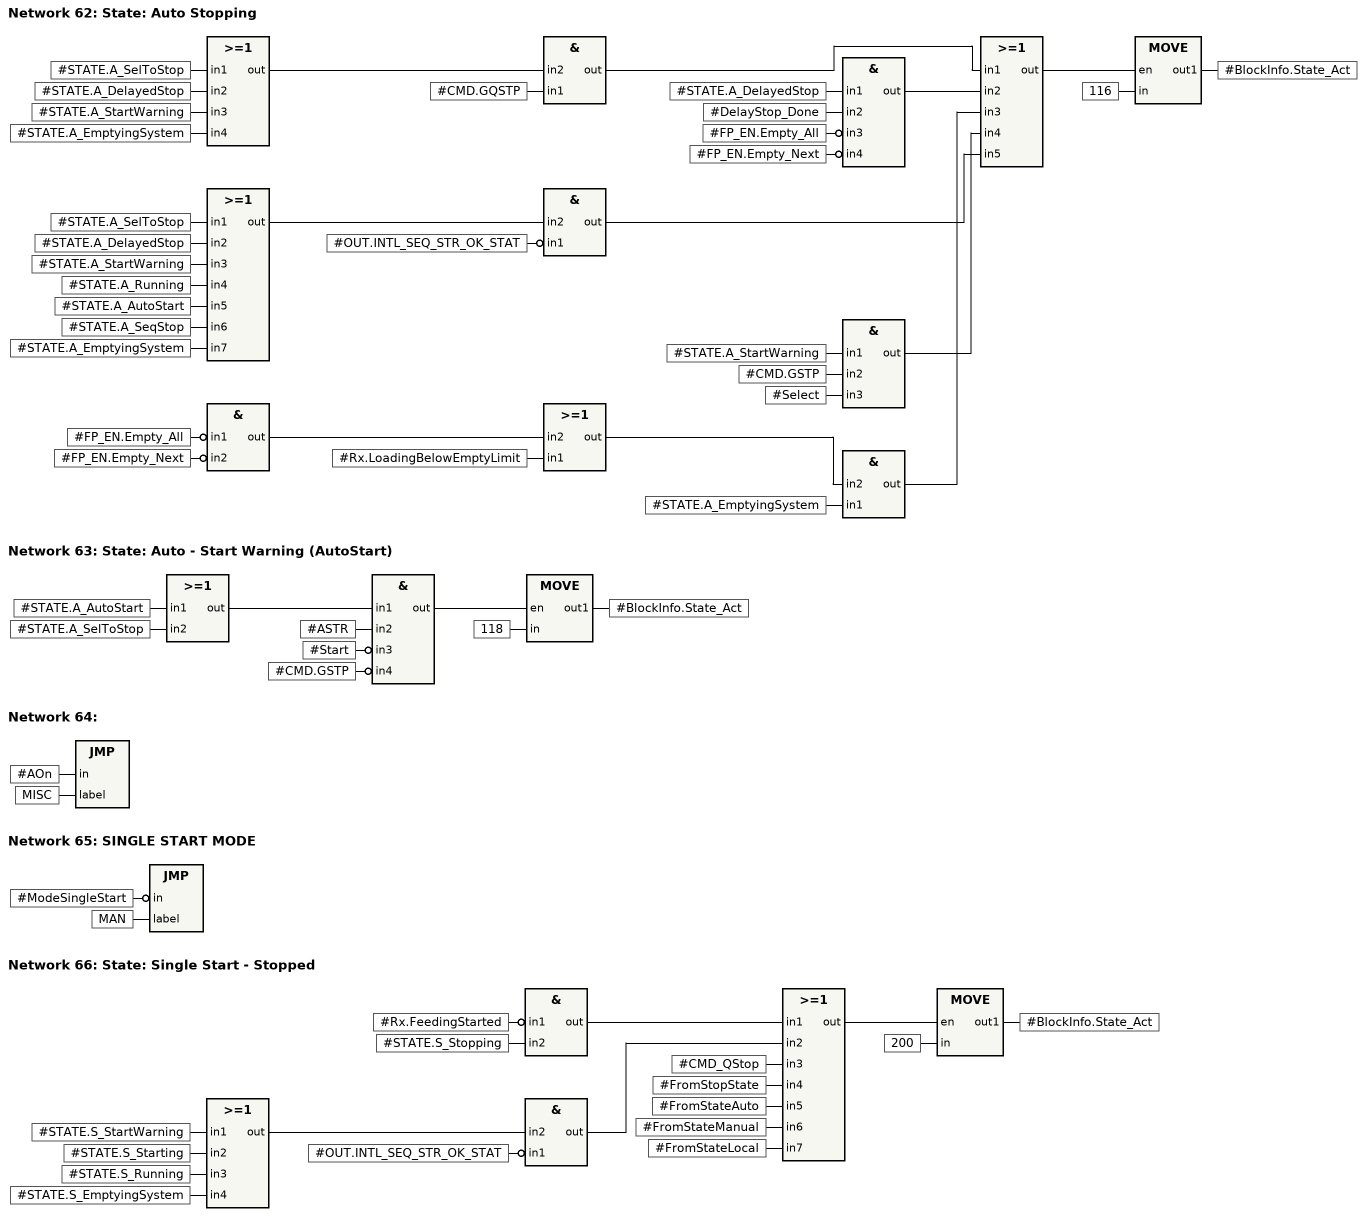
   IF ((#STATE.A_SelToStop OR #STATE.A_DelayedStop OR #STATE.A_StartWarning OR #STATE.A_EmptyingSystem) AND #CMD.GQSTP) OR (#STATE.A_DelayedStop AND #DelayStop_Done AND NOT #FP_EN.Empty_All AND NOT #FP_EN.Empty_Next) OR (((NOT #FP_EN.Empty_All AND NOT #FP_EN.Empty_Next) OR #Rx.LoadingBelowEmptyLimit) AND #STATE.A_EmptyingSystem) OR (#STATE.A_StartWarning AND #CMD.GSTP AND #Select) OR ((#STATE.A_SelToStop OR #STATE.A_DelayedStop OR #STATE.A_StartWarning OR #STATE.A_Running OR #STATE.A_AutoStart OR #STATE.A_SeqStop OR #STATE.A_EmptyingSystem) AND NOT #OUT.INTL_SEQ_STR_OK_STAT) THEN
       #BlockInfo.State_Act := 116;
   END_IF;
END_REGION

REGION Network 63: State: Auto - Start Warning (AutoStart)
   IF (#STATE.A_AutoStart OR #STATE.A_SelToStop) AND #ASTR AND NOT #Start AND NOT #CMD.GSTP THEN
       #BlockInfo.State_Act := 118;
   END_IF;
END_REGION

REGION Network 64
   IF #AOn THEN GOTO MISC; END_IF;
END_REGION

REGION Network 65: SINGLE START MODE
   SS1:
   IF NOT #ModeSingleStart THEN GOTO MAN; END_IF;
END_REGION

REGION Network 66: State: Single Start - Stopped
   IF (NOT #Rx.FeedingStarted AND #STATE.S_Stopping) OR ((#STATE.S_StartWarning OR #STATE.S_Starting OR #STATE.S_Running OR #STATE.S_EmptyingSystem) AND NOT #OUT.INTL_SEQ_STR_OK_STAT) OR #CMD_QStop OR #FromStopState OR #FromStateAuto OR #FromStateManual OR #FromStateLocal THEN
       #BlockInfo.State_Act := 200;
   END_IF;
END_REGION

REGION Network 67: State: Single Start - Start Warning
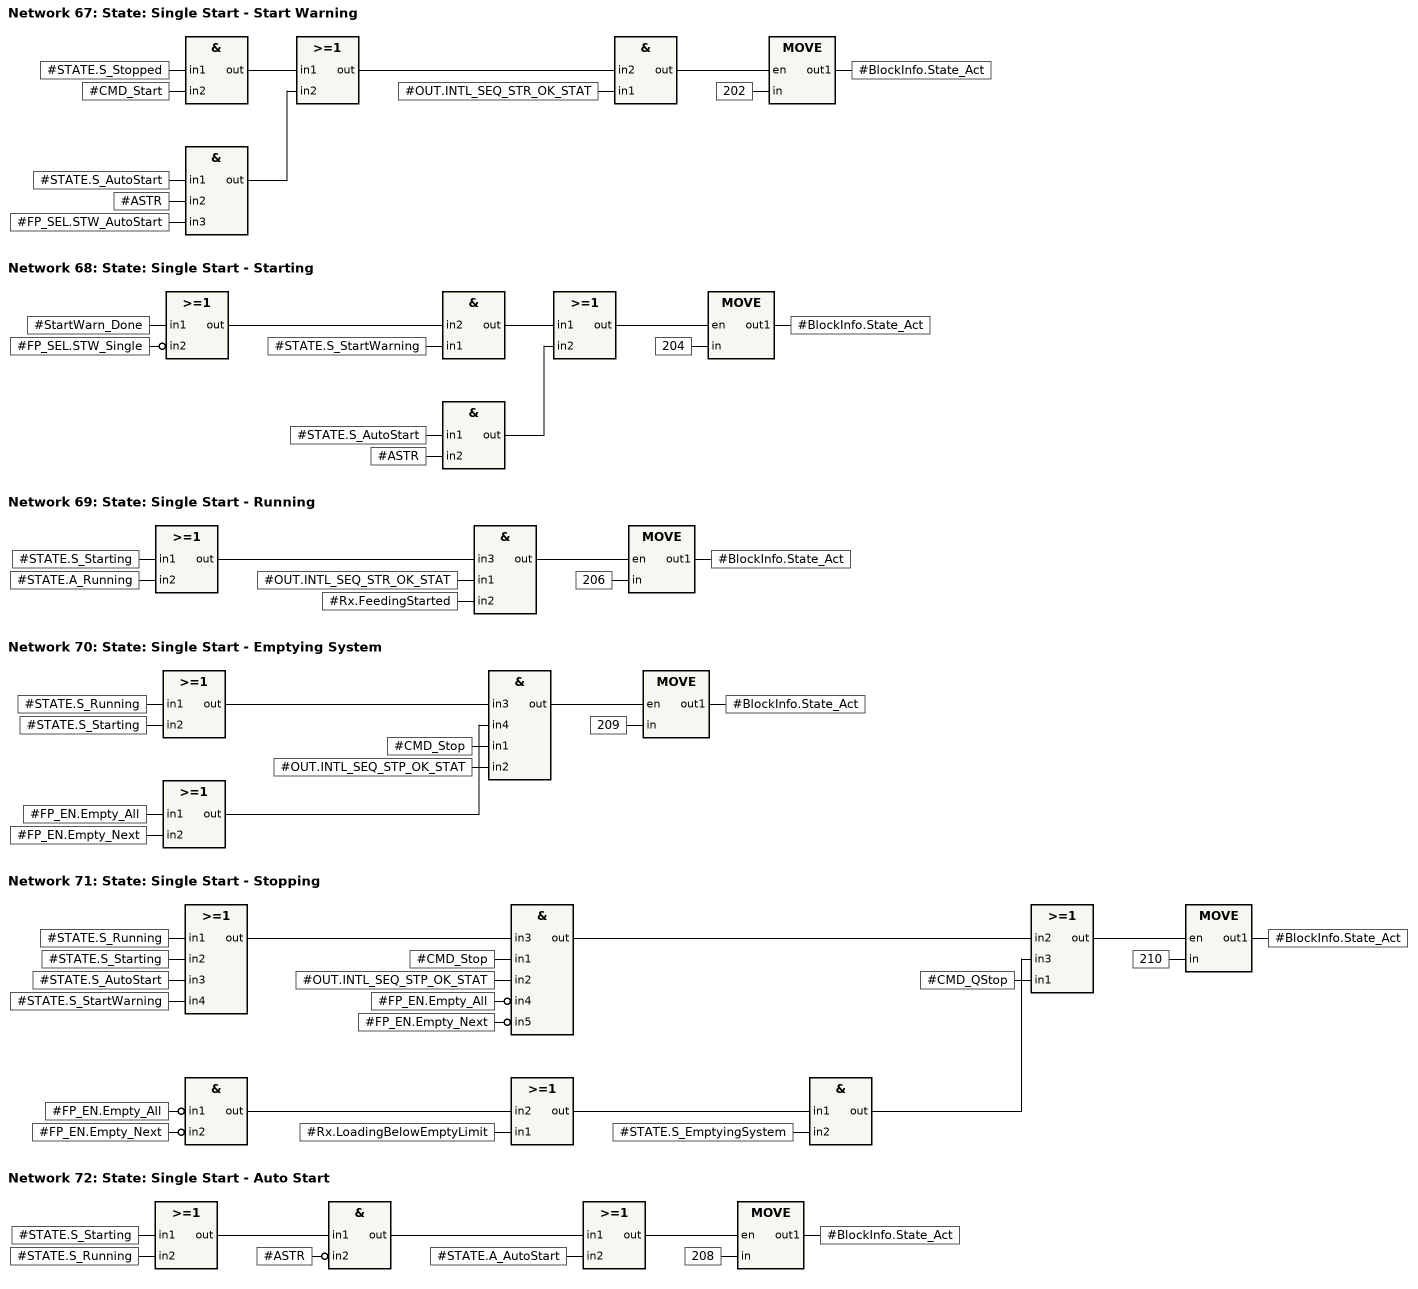
   IF ((#STATE.S_Stopped AND #CMD_Start) OR (#STATE.S_AutoStart AND #ASTR AND #FP_SEL.STW_AutoStart)) AND #OUT.INTL_SEQ_STR_OK_STAT THEN
       #BlockInfo.State_Act := 202;
   END_IF;
END_REGION

REGION Network 68: State: Single Start - Starting
   IF ((#StartWarn_Done OR NOT #FP_SEL.STW_Single) AND #STATE.S_StartWarning) OR (#STATE.S_AutoStart AND #ASTR) THEN
       #BlockInfo.State_Act := 204;
   END_IF;
END_REGION

REGION Network 69: State: Single Start - Running
   IF (#STATE.S_Starting OR #STATE.A_Running) AND #OUT.INTL_SEQ_STR_OK_STAT AND #Rx.FeedingStarted THEN
       #BlockInfo.State_Act := 206;
   END_IF;
END_REGION

REGION Network 70: State: Single Start - Emptying System
   IF (#STATE.S_Running OR #STATE.S_Starting) AND (#FP_EN.Empty_All OR #FP_EN.Empty_Next) AND #CMD_Stop AND #OUT.INTL_SEQ_STP_OK_STAT THEN
       #BlockInfo.State_Act := 209;
   END_IF;
END_REGION

REGION Network 71: State: Single Start - Stopping
   IF ((#STATE.S_Running OR #STATE.S_Starting OR #STATE.S_AutoStart OR #STATE.S_StartWarning) AND #CMD_Stop AND #OUT.INTL_SEQ_STP_OK_STAT AND NOT #FP_EN.Empty_All AND NOT #FP_EN.Empty_Next) OR (((NOT #FP_EN.Empty_All AND NOT #FP_EN.Empty_Next) OR #Rx.LoadingBelowEmptyLimit) AND #STATE.S_EmptyingSystem) OR #CMD_QStop THEN
       #BlockInfo.State_Act := 210;
   END_IF;
END_REGION

REGION Network 72: State: Single Start - Auto Start
   IF ((#STATE.S_Starting OR #STATE.S_Running) AND NOT #ASTR) OR #STATE.A_AutoStart THEN
       #BlockInfo.State_Act := 208;
   END_IF;
END_REGION

REGION Network 73
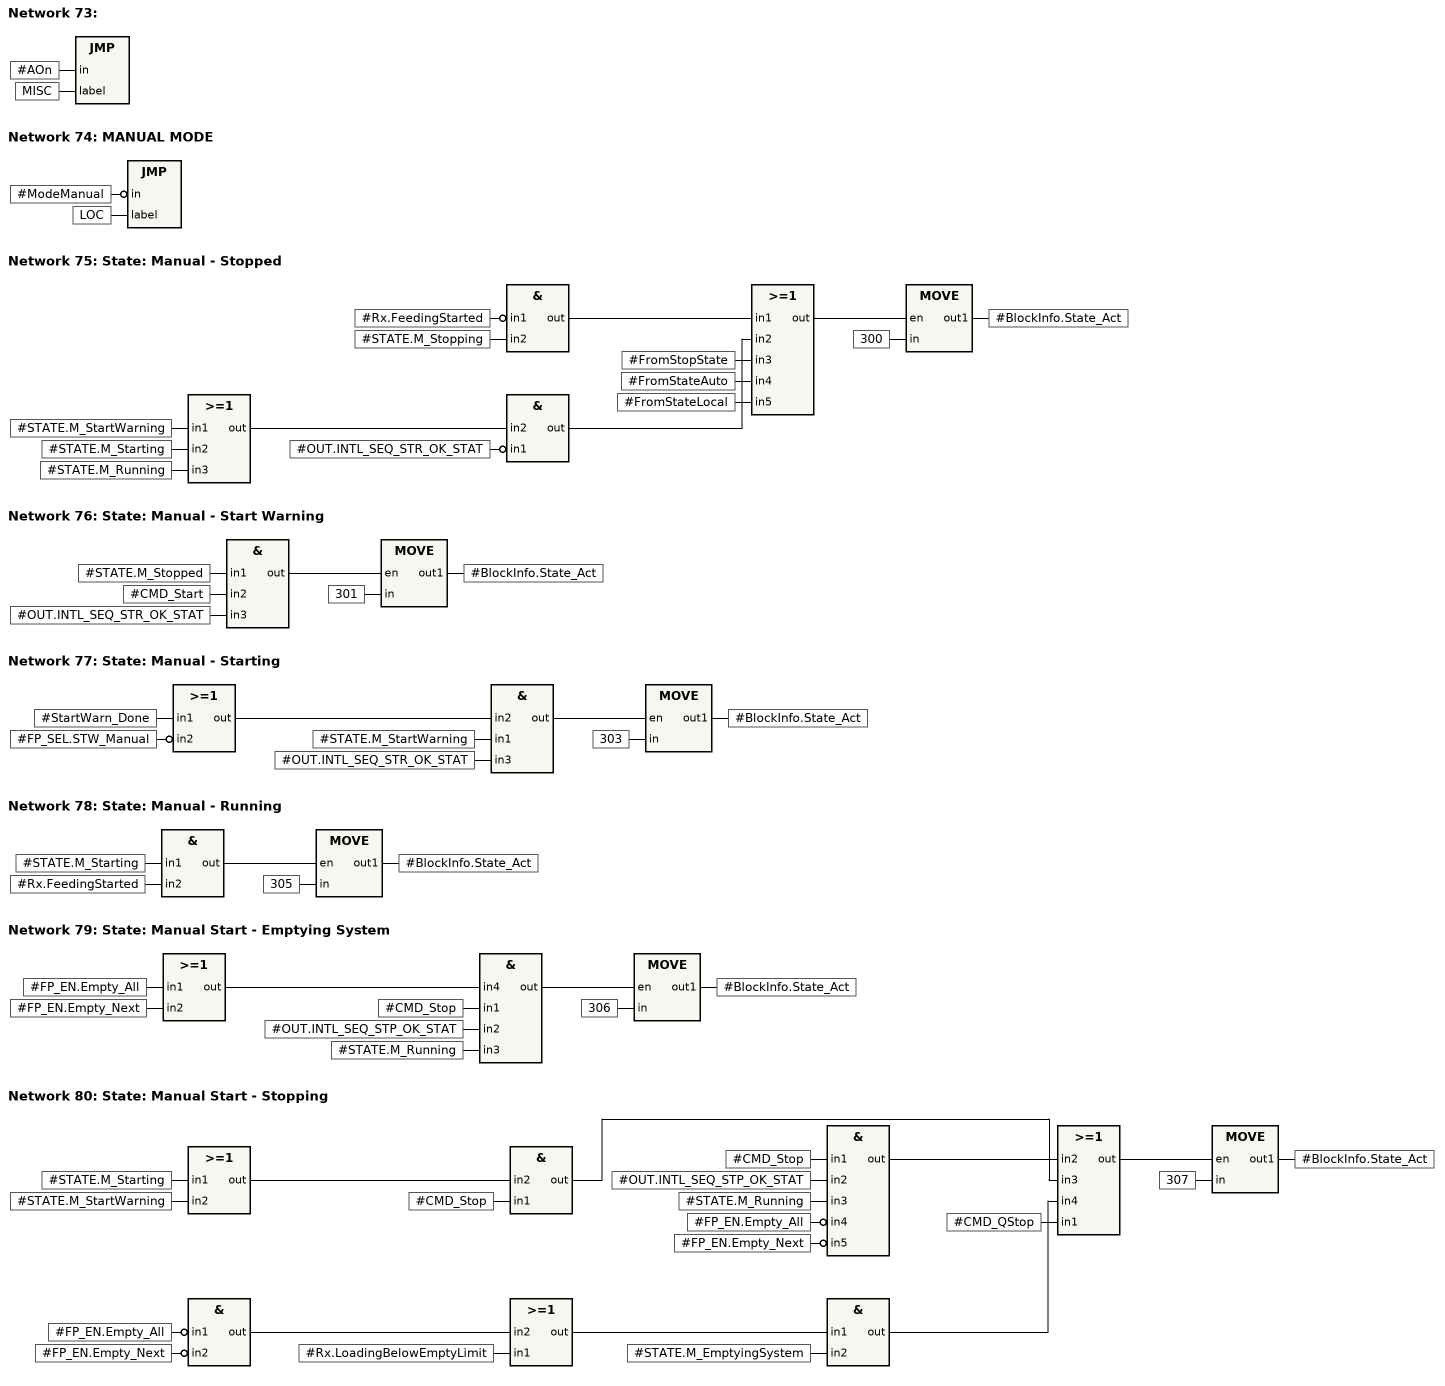
   IF #AOn THEN GOTO MISC; END_IF;
END_REGION

REGION Network 74: MANUAL MODE
   MAN:
   IF NOT #ModeManual THEN GOTO LOC; END_IF;
END_REGION

REGION Network 75: State: Manual - Stopped
   IF (NOT #Rx.FeedingStarted AND #STATE.M_Stopping) OR ((#STATE.M_StartWarning OR #STATE.M_Starting OR #STATE.M_Running) AND NOT #OUT.INTL_SEQ_STR_OK_STAT) OR #FromStopState OR #FromStateAuto OR #FromStateLocal THEN
       #BlockInfo.State_Act := 300;
   END_IF;
END_REGION

REGION Network 76: State: Manual - Start Warning
   IF #STATE.M_Stopped AND #CMD_Start AND #OUT.INTL_SEQ_STR_OK_STAT THEN #BlockInfo.State_Act := 301; END_IF;
END_REGION

REGION Network 77: State: Manual - Starting
   IF (#StartWarn_Done OR NOT #FP_SEL.STW_Manual) AND #STATE.M_StartWarning AND #OUT.INTL_SEQ_STR_OK_STAT THEN
       #BlockInfo.State_Act := 303;
   END_IF;
END_REGION

REGION Network 78: State: Manual - Running
   IF #STATE.M_Starting AND #Rx.FeedingStarted THEN #BlockInfo.State_Act := 305; END_IF;
END_REGION

REGION Network 79: State: Manual Start - Emptying System
   IF (#FP_EN.Empty_All OR #FP_EN.Empty_Next) AND #CMD_Stop AND #OUT.INTL_SEQ_STP_OK_STAT AND #STATE.M_Running THEN
       #BlockInfo.State_Act := 306;
   END_IF;
END_REGION

REGION Network 80: State: Manual Start - Stopping
   IF (#CMD_Stop AND #OUT.INTL_SEQ_STP_OK_STAT AND #STATE.M_Running AND NOT #FP_EN.Empty_All AND NOT #FP_EN.Empty_Next) OR ((#STATE.M_Starting OR #STATE.M_StartWarning) AND #CMD_Stop) OR (((NOT #FP_EN.Empty_All AND NOT #FP_EN.Empty_Next) OR #Rx.LoadingBelowEmptyLimit) AND #STATE.M_EmptyingSystem) OR #CMD_QStop THEN
       #BlockInfo.State_Act := 307;
   END_IF;
END_REGION

REGION Network 81
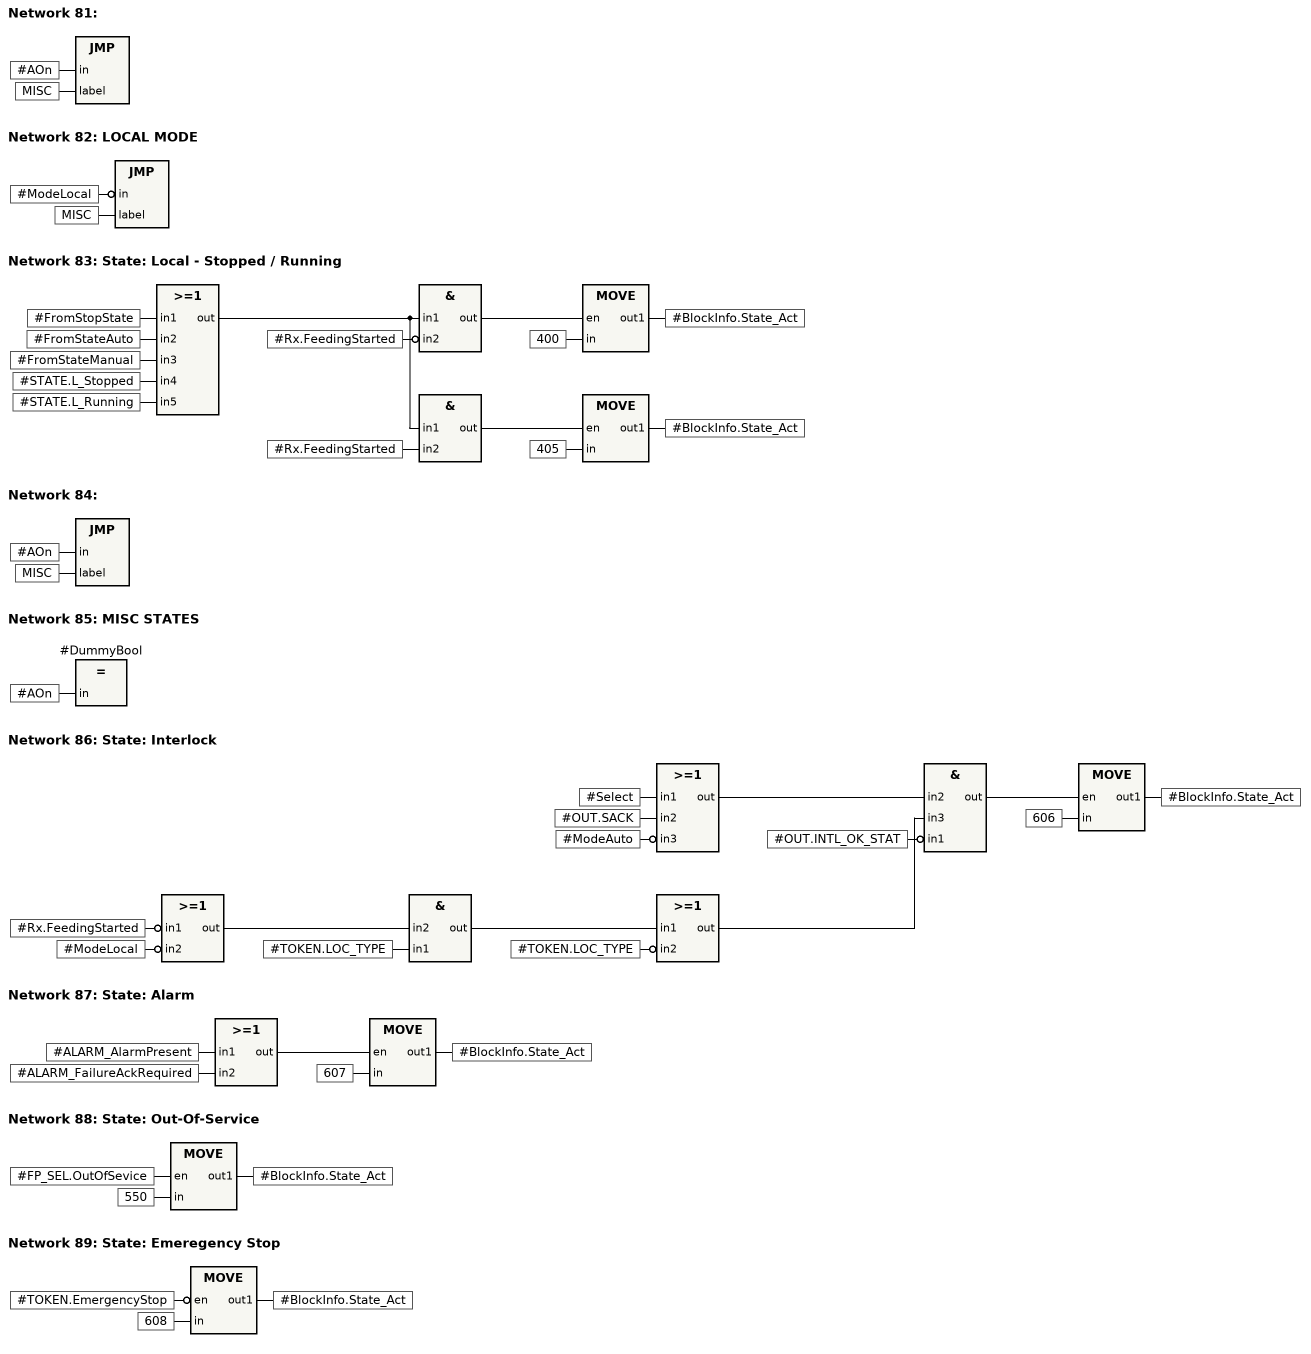
   IF #AOn THEN GOTO MISC; END_IF;
END_REGION

REGION Network 82: LOCAL MODE
   LOC:
   IF NOT #ModeLocal THEN GOTO MISC; END_IF;
END_REGION

REGION Network 83: State: Local - Stopped / Running
   #_w1 := #FromStopState OR #FromStateAuto OR #FromStateManual OR #STATE.L_Stopped OR #STATE.L_Running;
   IF #_w1 AND NOT #Rx.FeedingStarted THEN #BlockInfo.State_Act := 400; END_IF;
   IF #_w1 AND #Rx.FeedingStarted THEN #BlockInfo.State_Act := 405; END_IF;
END_REGION

REGION Network 84
   IF #AOn THEN GOTO MISC; END_IF;
END_REGION

REGION Network 85: MISC STATES
   MISC:
   #DummyBool := #AOn;
END_REGION

REGION Network 86: State: Interlock
   IF (#Select OR #OUT.SACK OR NOT #ModeAuto) AND (((NOT #Rx.FeedingStarted OR NOT #ModeLocal) AND #TOKEN.LOC_TYPE) OR NOT #TOKEN.LOC_TYPE) AND NOT #OUT.INTL_OK_STAT THEN
       #BlockInfo.State_Act := 606;
   END_IF;
END_REGION

REGION Network 87: State: Alarm
   IF #ALARM_AlarmPresent OR #ALARM_FailureAckRequired THEN #BlockInfo.State_Act := 607; END_IF;
END_REGION

REGION Network 88: State: Out-Of-Service
   IF #FP_SEL.OutOfSevice THEN #BlockInfo.State_Act := 550; END_IF;
END_REGION

REGION Network 89: State: Emeregency Stop
   IF NOT #TOKEN.EmergencyStop THEN #BlockInfo.State_Act := 608; END_IF;
END_REGION

REGION Network 90: SET STATE FLAGS - Auto Stopped
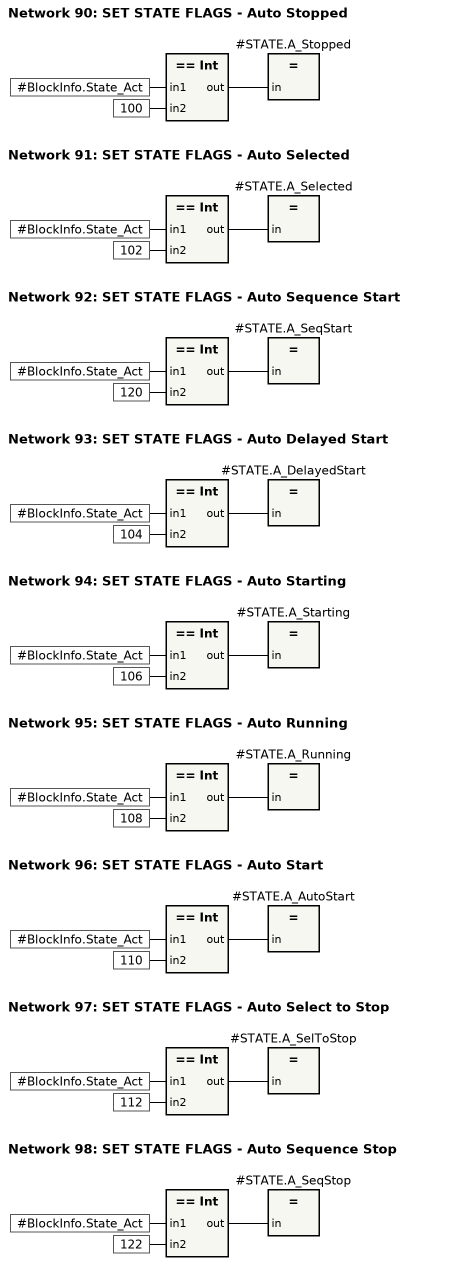
   #STATE.A_Stopped := #BlockInfo.State_Act = 100;
END_REGION

REGION Network 91: SET STATE FLAGS - Auto Selected
   #STATE.A_Selected := #BlockInfo.State_Act = 102;
END_REGION

REGION Network 92: SET STATE FLAGS - Auto Sequence Start
   #STATE.A_SeqStart := #BlockInfo.State_Act = 120;
END_REGION

REGION Network 93: SET STATE FLAGS - Auto Delayed Start
   #STATE.A_DelayedStart := #BlockInfo.State_Act = 104;
END_REGION

REGION Network 94: SET STATE FLAGS - Auto Starting
   #STATE.A_Starting := #BlockInfo.State_Act = 106;
END_REGION

REGION Network 95: SET STATE FLAGS - Auto Running
   #STATE.A_Running := #BlockInfo.State_Act = 108;
END_REGION

REGION Network 96: SET STATE FLAGS - Auto Start
   #STATE.A_AutoStart := #BlockInfo.State_Act = 110;
END_REGION

REGION Network 97: SET STATE FLAGS - Auto Select to Stop
   #STATE.A_SelToStop := #BlockInfo.State_Act = 112;
END_REGION

REGION Network 98: SET STATE FLAGS - Auto Sequence Stop
   #STATE.A_SeqStop := #BlockInfo.State_Act = 122;
END_REGION

REGION Network 99: SET STATE FLAGS - Auto Delayed Stop
